      U     "IX_U_AXIS_ALM_CDE_BIT_3"; //E ;BOOL;U-Achse Alarm Bit 3
      =     "I_WK_ALARMCODE_BIT_3"; //M     374.3;BOOL;M-EINGANG: KometU-Achse:Alarmcode Bit 2e3

      U     "IX_U_AXIS_CONFIRM"; //E ;BOOL;U-Achse Quittierung
      =     "I_WK_QUIT_KOMMANDO"; //M     374.4;BOOL;M-EINGANG: KometU-Achse:Quit bei Pt

      U     "IX_U_AXIS_ALARM_N"; //E ;BOOL;U-Achse kein Alarm
      =     "I_WK_NEG_ALARM"; //M     374.5;BOOL;M-EINGANG: KometU-Achse:Alar

      U     "IX_U_AXIS_TOOL_ACTIVE_N"; //E ;BOOL;U-Achse keine Bearbeitung
      =     "I_WK_NEG_WZ_AKTIV"; //M     374.6;BOOL;M-EINGANG: KometU-Achse:Werkzeug beschäftig

      U     "IX_U_AXIS_TOOL_READY"; //E ;BOOL;U-Achse Werkzeug Betriebsbereit
      =     "I_WK_WZ_BTB"; //M     374.7;BOOL;M-EINGANG: KometU-Achse:System bereit

      U     "IX_U_AXIS_REF_SIGNAL"; //E ;BOOL;U-Achse Referenzimpuls
      =     "I_WK_REF"; //M     375.0;BOOL;M-EINGANG: KometU-Achse:RefNocken

      U     "IX_U_AXIS_READY"; //E ;BOOL;U-Achse Achse Betriebsbereit
      =     "I_WK_BTB"; //M     375.1;BOOL;M-EINGANG: KometU-Achse:Achse bereit

      U     "IX_U_AXIS_SWITCH_PLUS"; //E ;BOOL;U-Achse Endschalter positiv
      =     "I_WK_ENDSCHALTER_PLUS"; //M     375.2;BOOL;M-EINGANG: KometU-Achse:Vorendschalter positiv

      U     "IX_U_AXIS_SWITCH_MINUS"; //E ;BOOL;U-Achse Endschalter negativ
      =     "I_WK_ENDSCHALTER_MINUS"; //M     375.3;BOOL;M-EINGANG: KometU-Achse:Vorendschalter negativ
NETWORK
TITLE =Eingaenge Nicht verwendete Eingänge
//Eingänge, die in der HW konfiguriert werden müssen, aber noch nicht verwendet
//werden.
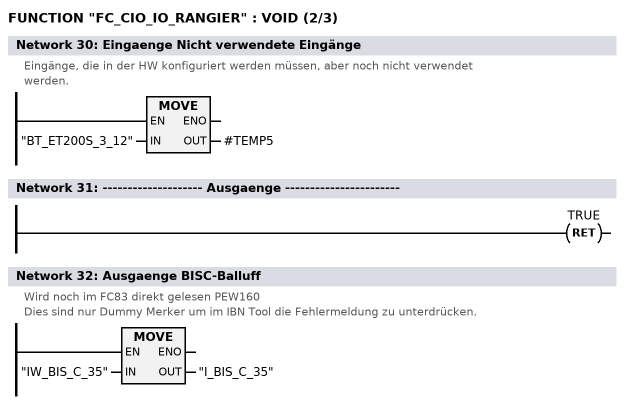
      L     "BT_ET200S_3_12"; //EW ;WORD;E5-03.5 Analogeingang Reserve
      T     #TEMP5;
NETWORK
TITLE =-------------------- Ausgaenge -----------------------

      BEA   ;

NETWORK
TITLE =Ausgaenge BISC-Balluff
//Wird noch im FC83 direkt gelesen PEW160
//Dies sind nur Dummy Merker um im IBN Tool die Fehlermeldung zu unterdrücken.
//
      L     "IW_BIS_C_35"; //PEW  1060;WORD;
      T     "I_BIS_C_35"; //MW    488;WORD;MW-EINGÄNGE:

NETWORK
TITLE =Ausgaenge allgemein
//Ausgänge
//
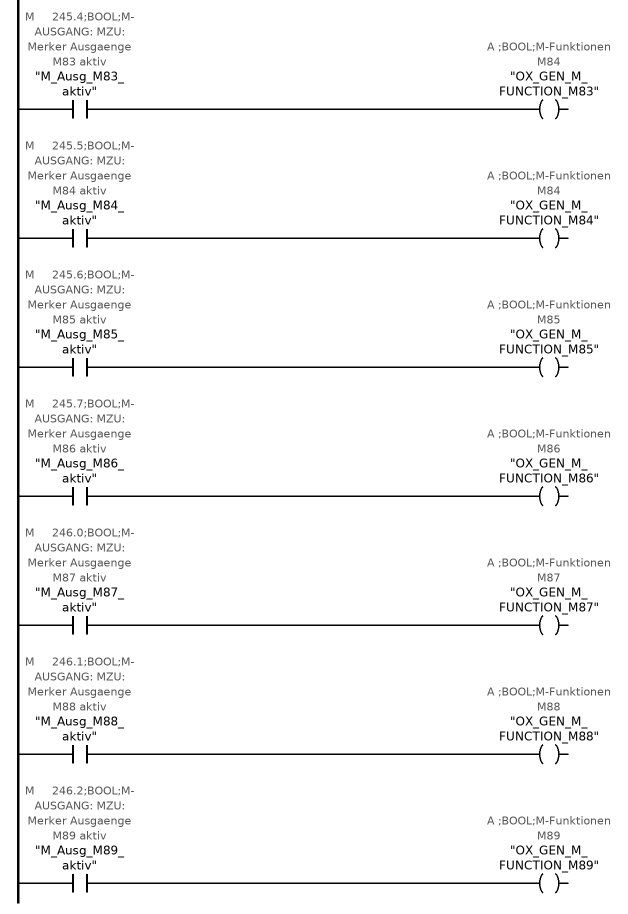
M003: NOP   0;

      U     "O_PW_FREIGABE"; //M     437.4;BOOL;M-AUSGANG: Anforderung Freigabe Palettenwechsel
      =     "OX_PC_ENABLE"; //A ;BOOL;Anforderung Freigabe Palettenwechsler   /G1-05.4

      U     "O_AL_PLC_BTB"; //M     432.1;BOOL;M-AUSGANG: Maschine 'Ein'  (CNC PLC Betriebsbereit)
      =     "OX_GEN_PLC_RDY"; //A ;BOOL;Maschine 'Ein'  (CNC PLC Betriebsbereit)

      U     "O_AL_Manual_Betrieb"; //M     432.2;BOOL;M-AUSGANG: Handbetrieb (Manual)
      =     "OX_AL_Manual_Betrieb"; //A ;BOOL;Handbetrieb (Manual)

      U     "O_GEN_CNC_PGM_ACTIVE"; //M     446.7;BOOL;M-AUSGANG: Betriebsstundenzaehler Programm laeuft
      =     "OX_GEN_CNC_PGM_ACTIVE"; //A ;BOOL;Betriebsstundenzaehler Programm laeuft

      U     "O_AL_XACHS_Bremse_auf"; //M     140.1;BOOL;M-AUSGANG: Ansteuerung Motorbremse X-Achse
      =     "OX_AL_XACHS_Bremse_auf"; //A ;BOOL;Ansteuerung Motorbremse X-Achse

      U     "O_AL_YACHS_Bremse_auf"; //M     140.3;BOOL;M-AUSGANG: Ansteuerung Motorbremse Y-Achse
      =     "OX_AL_YACHS_Bremse_auf"; //A ;BOOL;Ansteuerung Motorbremse Y-Achse

      U     "O_AL_ZACHS_Bremse_auf"; //M     140.5;BOOL;M-AUSGANG: Ansteuerung Motorbremse Z-Achse
      =     "OX_AL_ZACHS_Bremse_auf"; //A ;BOOL;Ansteuerung Motorbremse Z-Achse

      U     "O_AL_4ACHS_Bremse_auf"; //M     140.7;BOOL;M-AUSGANG: Ansteuerung Motorbremse 4-Achse
      =     "OX_AL_4ACHS_Bremse_auf"; //A ;BOOL;Ansteuerung Motorbremse 4-Achse

      U     "O_AL_5ACHS_Bremse_auf"; //M     141.1;BOOL;M-AUSGANG: Ansteuerung Motorbremse 5-Achse
      =     "OX_AL_5ACHS_Bremse_auf"; //A ;BOOL;Ansteuerung Motorbremse 5-Achse

      UN    "O_4_Klem_Bremse_Auf"; //M     433.5;BOOL;M-AUSGANG: 4.Achse Klemmung lösen
      =     "OX_AL_4ACHS_Klemmen"; //A ;BOOL;4.Achse klemmen

      UN    "O_5_Klem_Bremse_Auf"; //M     433.6;BOOL;M-AUSGANG: 5.Achse Klemmung lösen
      =     "OX_GEN_AXIS5_CLAMP"; //A ;BOOL;5.Achse klemmen

      UN    "O_5_Klem_Bremse_Auf"; //M     433.6;BOOL;M-AUSGANG: 5.Achse Klemmung lösen
      =     "OX_DH_CLAMP_RELEASE"; //A ;BOOL;Klemmung loesen NC-Teilapparat

      U     "M_SBH_AKTIV_ARBEITSRAUM"; //M     539.0;BOOL;SAFETY: SBH aktiv -> Freigabe Arbeitsraumtüre entriegeln
      =     "OX_GEN_CABIN_UNLOCK"; //A ;BOOL;Magnetverriegelung Kabinentüre entriegeln

      U     "O_AL_Hydraulik_Ein"; //M     433.3;BOOL;M-AUSGANG: Hydraulik 'Ein'
      =     "OX_GEN_HYD_ON"; //A ;BOOL;Hydraulik 'Ein'

      U     "O_AL_Druckluft_ein"; //M     433.2;BOOL;M-AUSGANG: Pneumatik 'Ein'
      =     "OX_GEN_CAIR_ON"; //A ;BOOL;Pneumatik 'Ein'

      U     "O_AL_Blasluft_M25"; //M     439.4;BOOL;M-AUSGANG: Blasluft Kuehlung Werkzeug 'Ein'
      =     "OX_SPI_CAIR_JETS_EXT"; //A ;BOOL;Blasluft Kuehlung Werkzeug 'Ein'

      U     "O_AL_4_BA_Selbsthaltung"; //M     437.7;BOOL;M-AUSGANG: Energiefreigabe 4.Betriebsart
      =     "OX_GEN_OM_4_ENABLE"; //A ;BOOL;Energiefreigabe 4.Betriebsart

      U     "O_AL_SCH_Pumpe_ein"; //M     432.4;BOOL;M-AUSGANG: Schmierung Maschine 'Ein'
      =     "OX_GEN_LUB_ON"; //A ;BOOL;Schmierung Maschine 'Ein'

      U     "O_AL_SCH_M26_Pumpe_ein"; //M     451.1;BOOL;M-AUSGANG: Dreh-Duchführung Ansteuerung Schmierpumpe 'Ein'
      =     "OX_SPI_ROTRA_LUB_ON"; //A ;BOOL;Dreh-Duchführung Ansteuerung Schmierpumpe 'Ein'

      U     "O_WZ_MIN_SCH_Ums_M7"; //M     104.7;BOOL;M-AUSGANG: Umschaltung Ventil Schmiersystem innere Kuehlmittelzufuhr
      =     "OX_TOOL_MQL_M7"; //A ;BOOL;Umschaltung Ventil Schmiersystem innere Kuehlmittelzufuhr

      U     "O_WZ_MIN_SCH_MV2"; //M      83.3;BOOL;M-AUSGANG: Minimalmengen Schmierung Ventil 2 Ein
      =     "OX_TOOL_MQL_VAL_2"; //A ;BOOL;Minimalmengen Schmierung Ventil 2 Ein

      U     "O_WZ_MIN_SCH_MV1"; //M     450.7;BOOL;M-AUSGANG: Minimalmengen Schmierung Ventil 1 Ein
      =     "OX_TOOL_MQL_VAL_1"; //A ;BOOL;Minimalmengen Schmierung Ventil 1 Ein

      U     "O_WZ_MIN_SCH_Ums_M8"; //M     104.2;BOOL;M-AUSGANG: Umschaltung Ventil Schmiersystem Kuehlmittel 1
      =     "OX_TOOL_MQL_M8"; //A ;BOOL;Umschaltung Ventil Schmiersystem Kuehlmittel 1

      U     "O_AL_Tempkomp_DSR"; //M     432.5;BOOL;M-AUSGANG: Temperaturkompensation rücksetzen Synchronisation Temperaturdaten
      =     "OX_AL_Tempkomp_DSR"; //A ;BOOL;TEMPERATURKOMPENSATION: rücksetzen Synchronisation Temperaturdaten

      U     "O_AL_Tempkomp_CTS"; //M     432.6;BOOL;M-AUSGANG: Temperaturkompensation   Temperaturdaten auslesen
      =     "OX_AL_Tempkomp_CTS"; //A ;BOOL;TEMPERATURKOMPENSATION: Temperaturdaten auslesen

      U     "O_AL_LM_RD"; //M     327.0;BOOL;M-AUSGANG: Signalleuchte Farbe RD
      =     "OX_GEN_SIGNALLAMP_RD"; //A ;BOOL;Signalleuchte Farbe RD

      U     "O_AL_LM_GN"; //M     327.2;BOOL;M-AUSGANG: Signalleuchte Farbe GN
      =     "OX_GEN_SIGNALLAMP_GN"; //A ;BOOL;Signalleuchte Farbe GN

      U     "O_AL_LM_YE"; //M     327.1;BOOL;M-AUSGANG: Signalleuchte Farbe YE
      =     "OX_GEN_SIGNALLAMP_YE"; //A ;BOOL;Signalleuchte Farbe YE

      U     "O_AL_LM_BU"; //M     327.3;BOOL;M-AUSGANG: Signalleuchte Farbe BU
      =     "OX_GEN_SIGNALLAMP_BU"; //A ;BOOL;Signalleuchte Farbe BU

      U     "O_GEN_OM_ID_DATA_0"; //M     446.5;BOOL;M-AUSGANG: Smartkey -  Rückmeldung Daten-Spur 1
      =     "OX_GEN_OM_ID_DATA_0"; //A ;BOOL;Smartkey: Rückmeldung Daten – Spur 1

      U     "O_GEN_OM_ID_DATA_1"; //M     446.6;BOOL;M-AUSGANG: Smartkey -  Rückmeldung Daten-Spur 2
      =     "OX_GEN_OM_ID_DATA_1"; //A ;BOOL;Smartkey: Rückmeldung Daten – Spur 2

      U     "O_GEN_OPTWAVE_GN"; //M    2061.2;BOOL;M-AUSGANG: Signalband Farbe Grün
      =     "OX_GEN_OPTWAVE_GN"; //A ;BOOL;Signalband neues Design Farbe GN

      U     "O_GEN_OPTWAVE_RD"; //M    2061.0;BOOL;M-AUSGANG: Signalband Farbe Rot
      =     "OX_GEN_OPTWAVE_RD"; //A ;BOOL;Signalband neues Design Farbe RD

      U     "O_GEN_OPTWAVE_BU"; //M    2061.3;BOOL;M-AUSGANG: Signalband Farbe Blau
      =     "OX_GEN_OPTWAVE_BU"; //A ;BOOL;Signalband neues Design Farbe  BU

      U     "O_AL_Start_Sig_Renishaw"; //M     433.7;BOOL;M-AUSGANG: Messtasterfreigabe
      =     "OX_AL_Start_Sig_Renishaw"; //A ;BOOL;Messtasterfreigabe

      U     "O_AL_Start_Sig_Renishaw"; //M     433.7;BOOL;M-AUSGANG: Messtasterfreigabe
      =     "OX_TP_ENABLE"; //A ;BOOL;Startsignal Messtaster

      U     "O_AL_NEBELABSCH_EIN"; //M     113.6;BOOL;M-AUSGANG: Nebel- u.Rauchabscheider 'Ein'
      =     "OX_OMS_ON"; //A ;BOOL;Nebel- u.Rauchabscheider 'Ein'

      U     "O_AL_NEG_POWERSAVE_STBY"; //M     344.7;BOOL;M-AUSGANG: Maschinenabschaltung
      =     "OX_GEN_POWERSAVE_N"; //A ;BOOL;Maschinenabschaltung

      U     "O_PW_SPANNDRUCK_HYD_AUS"; //M     436.3;BOOL;M-AUSGANG: MA H4-03.7 Spannvorrichtung Verriegelung Palettenwechsler
      =     "OX_PC_CL_PRESS_HYD_OFF"; //A ;BOOL;MA H4-03.7 Spannvorrichtung Verriegelung Palettenwechs

      U     "O_Funktion_M20"; //M     435.6;BOOL;M-AUSGANG: Zusatzfunktion M190
      =     "OX_AL_Funktion_M20"; //A ;BOOL;M-Funktionen M190

      U     "M_Ausg_M80_aktiv"; //M     245.1;BOOL;M-AUSGANG: MZU: Merker Ausgaenge M80 aktiv
      =     "OX_GEN_M_FUNCTION_M80"; //A ;BOOL;M-Funktionen M80

      U     "M_Ausg_M81_aktiv"; //M     245.2;BOOL;M-AUSGANG: MZU: Merker Ausgaenge M81 aktiv
      =     "OX_GEN_M_FUNCTION_M81"; //A ;BOOL;M-Funktionen M81

      U     "M_Ausg_M82_aktiv"; //M     245.3;BOOL;M-AUSGANG: MZU: Merker Ausgaenge M82 aktiv
      =     "OX_GEN_M_FUNCTION_M82"; //A ;BOOL;M-Funktionen M82

      U     "M_Ausg_M83_aktiv"; //M     245.4;BOOL;M-AUSGANG: MZU: Merker Ausgaenge M83 aktiv
      =     "OX_GEN_M_FUNCTION_M83"; //A ;BOOL;M-Funktionen M84

      U     "M_Ausg_M84_aktiv"; //M     245.5;BOOL;M-AUSGANG: MZU: Merker Ausgaenge M84 aktiv
      =     "OX_GEN_M_FUNCTION_M84"; //A ;BOOL;M-Funktionen M84

      U     "M_Ausg_M85_aktiv"; //M     245.6;BOOL;M-AUSGANG: MZU: Merker Ausgaenge M85 aktiv
      =     "OX_GEN_M_FUNCTION_M85"; //A ;BOOL;M-Funktionen M85

      U     "M_Ausg_M86_aktiv"; //M     245.7;BOOL;M-AUSGANG: MZU: Merker Ausgaenge M86 aktiv
      =     "OX_GEN_M_FUNCTION_M86"; //A ;BOOL;M-Funktionen M86

      U     "M_Ausg_M87_aktiv"; //M     246.0;BOOL;M-AUSGANG: MZU: Merker Ausgaenge M87 aktiv
      =     "OX_GEN_M_FUNCTION_M87"; //A ;BOOL;M-Funktionen M87

      U     "M_Ausg_M88_aktiv"; //M     246.1;BOOL;M-AUSGANG: MZU: Merker Ausgaenge M88 aktiv
      =     "OX_GEN_M_FUNCTION_M88"; //A ;BOOL;M-Funktionen M88

      U     "M_Ausg_M89_aktiv"; //M     246.2;BOOL;M-AUSGANG: MZU: Merker Ausgaenge M89 aktiv
      =     "OX_GEN_M_FUNCTION_M89"; //A ;BOOL;M-Funktionen M89
NETWORK
TITLE =Ausgänge für Vibrationssensor

      L     "DB_PLC_MD_DB20".UDInt._044_ANWAHL_VIBRATIONSEN;
      L     1;
      >=I   ;
      SPBN  kVMS;

      L     "MW_VMS_SPI_SPEED_RPM"; //MW    612;INT;Analogausgang Vibrationssensor Spindeldrehzahl
      T     "OW_VMS_SPI_SPEED_RPM"; //AW ;WORD;

      U     "O_VMS_MSG_BEA_START"; //M     671.2;BOOL;
      =     "OX_VMS_MSG_BEA_START"; //A ;BOOL;

kVMS: NOP   0;
NETWORK
TITLE =Ausgaenge an NCU und NC Baugruppe SOLUTIONLINE
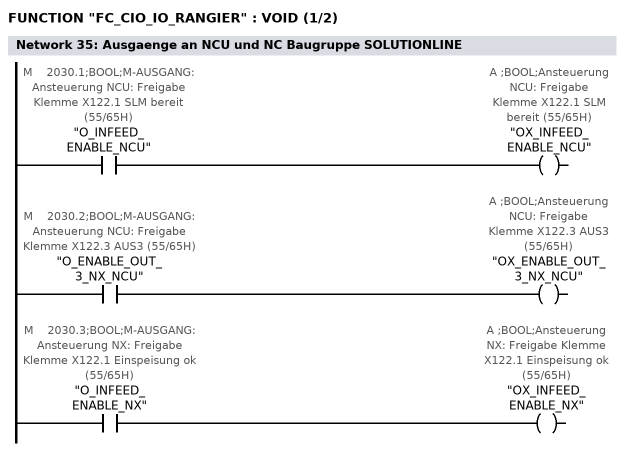

      NOP   0;

      U     "O_INFEED_ENABLE_NCU"; //M    2030.1;BOOL;M-AUSGANG: Ansteuerung NCU: Freigabe Klemme X122.1 SLM bereit (55/65H)
      =     "OX_INFEED_ENABLE_NCU"; //A ;BOOL;Ansteuerung NCU: Freigabe Klemme X122.1 SLM bereit (55/65H)

      U     "O_ENABLE_OUT_3_NX_NCU"; //M    2030.2;BOOL;M-AUSGANG: Ansteuerung NCU: Freigabe Klemme X122.3 AUS3 (55/65H)
      =     "OX_ENABLE_OUT_3_NX_NCU"; //A ;BOOL;Ansteuerung NCU: Freigabe Klemme X122.3 AUS3 (55/65H)

      U     "O_INFEED_ENABLE_NX"; //M    2030.3;BOOL;M-AUSGANG: Ansteuerung NX: Freigabe Klemme X122.1 Einspeisung ok (55/65H)
      =     "OX_INFEED_ENABLE_NX"; //A ;BOOL;Ansteuerung NX: Freigabe Klemme X122.1 Einspeisung ok (55/65H)
NETWORK
TITLE =Ausgaenge Schwenkkopf und Spindel
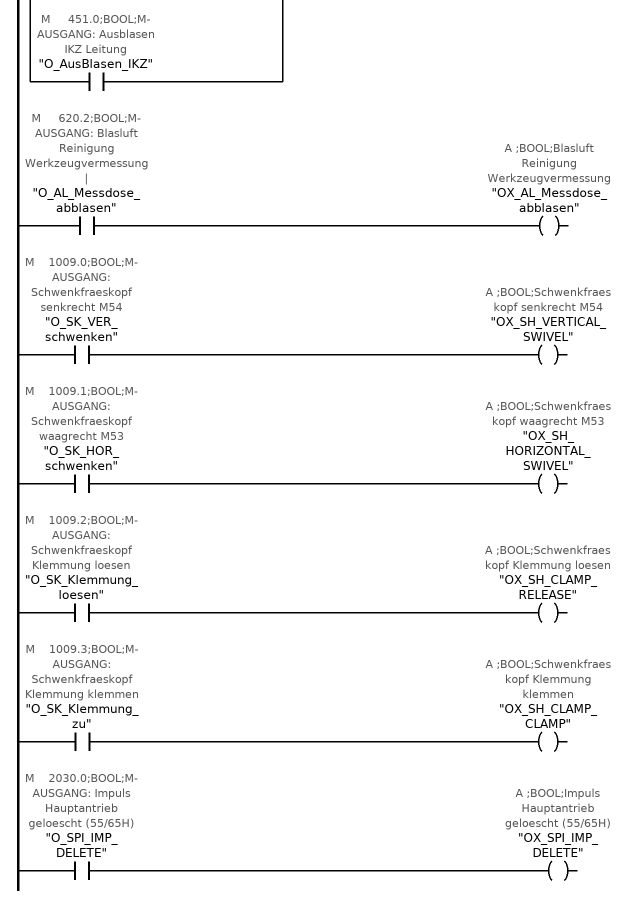

      U     "O_SPI_klemmen"; //M     283.1;BOOL;M-AUSGANG: Fraesspindel klemmen
      =     "OX_SPI_CLAMP"; //A ;BOOL;Fraesspindel klemmen

      U     "O_SPI_loesen"; //M     283.2;BOOL;M-AUSGANG: Fraesspindel loesen
      =     "OX_SPI_RELEASE"; //A ;BOOL;Fraesspindel loesen

      U     "O_Y_Umschaltung_SPI"; //M     447.1;BOOL;M-AUSGANG: Stern Dreieck: Ausgang Stern
      =     "OX_SPI_WYE"; //A ;BOOL;Stern Dreieck: Ausgang Stern

      U     "O_D_Umschaltung_SPI"; //M     447.2;BOOL;M-AUSGANG: Stern Dreieck: Ausgang Dreieck
      =     "OX_SPI_DELTA"; //A ;BOOL;Stern Dreieck: Ausgang Dreieck

      U     "O_SK_1_Stufe_Getriebe"; //M     433.0;BOOL;M-AUSGANG: Drehzahlschaltung Hauptantrieb mit Getriebe    Drehzahl kleiner
      =     "OX_SH_GEAR_STAGE1"; //A ;BOOL;Drehzahlschaltung Hauptantrieb mit Getriebe    Drehzahl kle

      U     "O_SK_2_Stufe_Getriebe"; //M     433.1;BOOL;M-AUSGANG: Drehzahlschaltung Hauptantrieb mit Getriebe    Drehzahl größer
      =     "OX_SH_GEAR_STAGE2"; //A ;BOOL;Drehzahlschaltung Hauptantrieb mit Getriebe    Drehzahl gr

      U     "O_SPI_SCH_LUFT"; //M     435.1;BOOL;M-AUSGANG: Schwenkfräskopf Druckluft Schmierung 'Ein'
      =     "OX_SPI_LUB_CAIR_ON"; //A ;BOOL;Schwenkfräskopf Druckluft Schmierung 'Ein'

      U     "O_SPI_SCH_OEL"; //M     435.0;BOOL;M-AUSGANG: Schmierung Hauptantrieb 24.000 U/min
      =     "OX_SPI_LUB_OIL_PUMP_ON"; //A ;BOOL;Schmierung Hauptantrieb 24.000 U/min

      U     "O_WZKegel_Blasluft"; //M     434.0;BOOL;M-AUSGANG: Messtaster Messstelle reinigen (M29) und  Werkzeugkegel ausblasen
      O(    ;
      U     "O_Blasluft_Messtaster"; //M     440.3;BOOL;M-AUSGANG: Blasluft Messtaster
      UN    "M_24aktiv"; //M     214.3;BOOL;LA: Laser ausfahren M24 aktiv
      )     ;
      O     "O_M7_Luftkuehlung"; //M     443.4;BOOL;M-AUSGANG: M7 Luftkuehlung
      O     "O_AusBlasen_IKZ"; //M     451.0;BOOL;M-AUSGANG: Ausblasen IKZ Leitung
      =     "OX_SPI_CAIR_TOOL"; //A ;BOOL;Druckluft Werkzeugkegel ausblasen

      U     "O_AL_Messdose_abblasen"; //M     620.2;BOOL;M-AUSGANG: Blasluft Reinigung Werkzeugvermessung |
      =     "OX_AL_Messdose_abblasen"; //A ;BOOL;Blasluft Reinigung Werkzeugvermessung

      U     "O_SK_VER_schwenken"; //M    1009.0;BOOL;M-AUSGANG: Schwenkfraeskopf senkrecht M54
      =     "OX_SH_VERTICAL_SWIVEL"; //A ;BOOL;Schwenkfraeskopf senkrecht M54

      U     "O_SK_HOR_schwenken"; //M    1009.1;BOOL;M-AUSGANG: Schwenkfraeskopf waagrecht M53
      =     "OX_SH_HORIZONTAL_SWIVEL"; //A ;BOOL;Schwenkfraeskopf waagrecht M53

      U     "O_SK_Klemmung_loesen"; //M    1009.2;BOOL;M-AUSGANG: Schwenkfraeskopf Klemmung loesen
      =     "OX_SH_CLAMP_RELEASE"; //A ;BOOL;Schwenkfraeskopf Klemmung loesen

      U     "O_SK_Klemmung_zu"; //M    1009.3;BOOL;M-AUSGANG: Schwenkfraeskopf Klemmung klemmen
      =     "OX_SH_CLAMP_CLAMP"; //A ;BOOL;Schwenkfraeskopf Klemmung klemmen

      U     "O_SPI_IMP_DELETE"; //M    2030.0;BOOL;M-AUSGANG: Impuls Hauptantrieb geloescht (55/65H)
      =     "OX_SPI_IMP_DELETE"; //A ;BOOL;Impuls Hauptantrieb geloescht (55/65H)

NETWORK
TITLE =Ausgänge WZ-Spanner

//Bei H-Maschinen werdem die Ausgänge durch den OB35 Aufruf geschrieben (Span_zu_Span_Zeit Optimierung)
      U     "DB_CONFIG".ANWAHL_DURCH_USER_DATA.MASCHTYP_3071_AKTIV;
      SPB   Hma2;

      U     "O_AL_WZ_Spanner_Loesen"; //M     433.4;BOOL;M-AUSGANG: Werkzeugspanner lösen (Autobetr)/Anwahl lösen (Handbetr)
      O     "M_O_Anwahl_WZS_Man"; //M     195.5;BOOL;WSP: Ausgang Manuelles loesen Spanner
      =     "OX_SPI_TL_CLAMP_RELEASE"; //A ;BOOL;Werkzeugspanner loesen

      UN    "O_AL_WZ_Spanner_Loesen"; //M     433.4;BOOL;M-AUSGANG: Werkzeugspanner lösen (Autobetr)/Anwahl lösen (Handbetr)
      UN    "M_Tast_Man_WZSp"; //M     386.0;BOOL;WZ-SPANNER:Werkzeugspanner manuell lösen
      =     "OX_SPI_TL_CLP_CLAMP"; //A ;BOOL;Werkzeugspanner spannen

Hma2: NOP   0;
NETWORK
TITLE =Ausgaenge Handrad
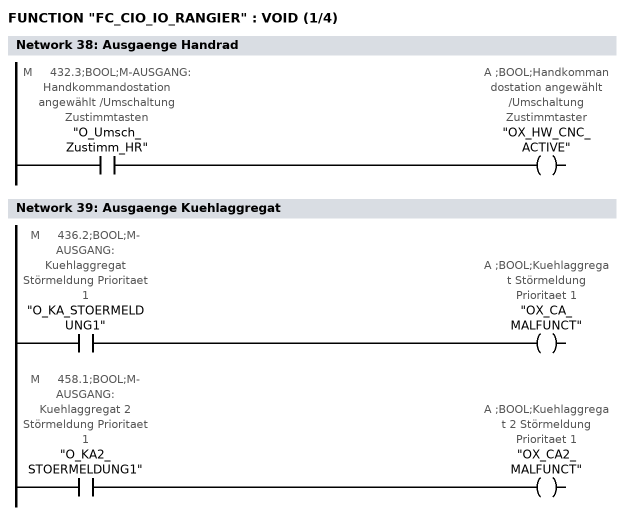

      NOP   0;

      U     "O_Umsch_Zustimm_HR"; //M     432.3;BOOL;M-AUSGANG: Handkommandostation angewählt /Umschaltung Zustimmtasten
      =     "OX_HW_CNC_ACTIVE"; //A ;BOOL;Handkommandostation angewählt /Umschaltung Zustimmtaster

NETWORK
TITLE =Ausgaenge Kuehlaggregat

      NOP   0;

      U     "O_KA_STOERMELDUNG1"; //M     436.2;BOOL;M-AUSGANG: Kuehlaggregat Störmeldung Prioritaet 1
      =     "OX_CA_MALFUNCT"; //A ;BOOL;Kuehlaggregat Störmeldung Prioritaet 1

      U     "O_KA2_STOERMELDUNG1"; //M     458.1;BOOL;M-AUSGANG: Kuehlaggregat 2 Störmeldung Prioritaet 1
      =     "OX_CA2_MALFUNCT"; //A ;BOOL;Kuehlaggregat 2 Störmeldung Prioritaet 1
NETWORK
TITLE =Ausgaenge Spannhydraulik
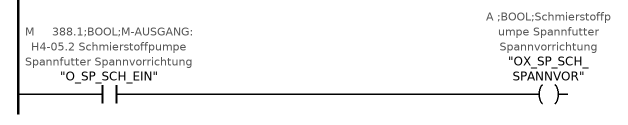

      NOP   0;

      U     "O_SP_HYD_EIN"; //M     458.3;BOOL;M-AUSGANG: Spannhydraulik Pumpe ein
      =     "OX_HCD_ON"; //A ;BOOL;Spannhydraulik ein   /H4-01.6

      U     "O_SP_HYD_RPL_LOESEDR_OK"; //M     382.0;BOOL;M-AUSGANG: Spannvorrichtung Loesedruck vorhanden
      =     "OX_HCD_CL_PR_SST_RELD_H"; //A ;BOOL;Spannhydraulik Leuchtmelder Vorrichtung entspannen   /H4-10.6

      U     "O_SP_HYD_RPL_SPANNDR_OK"; //M     382.1;BOOL;M-AUSGANG: Spannvorrichtung Spanndruck vorhanden
      =     "OX_HCD_CL_PR_SST_CLPED_H"; //A ;BOOL;Spannhydraulik Leuchtmelder Vorrichtung spannen   /H4-10.3

      U     "O_SP_H_SPANNSTELLE_1"; //M     356.0;BOOL;M-AUSGANG: Spannhydraulik Lampe Spannstelle 1
      =     "OX_HCD_SST_CL_PO_1_SEL_H"; //A ;BOOL;Spannhydraulik Rüstplatz Leuchtmelder Spannstelle 1 aktiv   /H4-50.3

      U     "O_SP_H_SPANNSTELLE_2"; //M     356.1;BOOL;M-AUSGANG: Spannhydraulik Lampe Spannstelle 2
      =     "OX_HCD_SST_CL_PO_2_SEL_H"; //A ;BOOL;Spannhydraulik Rüstplatz Leuchtmelder Spannstelle 2 aktiv   /H4-50.6

      U     "O_SP_H_SPANNSTELLE_3"; //M     356.2;BOOL;M-AUSGANG: Spannhydraulik Lampe Spannstelle 3
      =     "OX_SP_H_SPANNSTELLE_3"; //A ;BOOL;Spannhydraulik Lampe Spannstelle 3

      U     "O_SP_H_SPANNSTELLE_4"; //M     356.3;BOOL;M-AUSGANG: Spannhydraulik Lampe Spannstelle 4
      =     "OX_SP_H_SPANNSTELLE_4"; //A ;BOOL;Spannhydraulik Lampe Spannstelle 4

      U     "O_SST_FIXT_CL_PO_1_CLE"; //M     384.6;BOOL;MA H4-94.2 Auflagenkontrolle Luft für Reinigung (hoher ALK-Druck)
      =     "OX_SST_FIXT_CL_PO_1_CLE"; //A ;BOOL;H4-94.2 Auflagenkontrolle Luft für Reinigung (hoher ALK-Druck)

      U     "O_SST_SC_SENS_ACT"; //M     384.7;BOOL;MA H4-94.4 Auflagenkontrolle Luft für Messung (niedriger ALK-Druck)
      =     "OX_SST_SC_SENS_ACT"; //A ;BOOL;H4-94.4 Auflagenkontrolle Luft für Messung (niedriger ALK-Druck)

      U     "O_SST_SC_CL_PO_1_STATE"; //M     379.4;BOOL;MA H4-93.2 Status Auflagenkontrolle Spannstelle 1 (Meldeleuchte)
      =     "OX_SST_SC_CL_PO_1_STATE"; //A ;BOOL;H4-93.2 Status Auflagenkontrolle Spannstelle 1 (Meldeleuchte)

      U     "O_SST_SC_CL_PO_2_STATE"; //M     379.5;BOOL;MA H4-93.4 Status Auflagenkontrolle Spannstelle 2 (Meldeleuchte)
      =     "OX_SST_SC_CL_PO_2_STATE"; //A ;BOOL;H4-93.4 Status Auflagenkontrolle Spannstelle 2 (Meldeleuchte)

      U     "O_SP_RPL_BLASLUFT"; //M     357.7;BOOL;M-AUSGANG: Ventil Luft für Vorrichtung Abblasen
      =     "OX_HCD_SST_BLOW_AIR"; //A ;BOOL;Medienkupplung Ruestplatz abblasen

      U     "O_SP_MPL_BLASLUFT"; //M     205.7;BOOL;M-AUSGANG: Blasluft Medienkupplung Spannhydraulik 'Ein'
      =     "OX_HCD_TST_MCON_CLEAN"; //A ;BOOL;Hydraulik Maschinenplatz Kupplung abblasen   /H4-08.2

      U     "O_SP_RPL_MPL_BLASLUFT"; //M      24.6;BOOL;M-AUSGANG: Ventil Blasluft Medienkupplung
      =     "OX_SP_RPL_MPL_BLASLUFT"; //A ;BOOL;Ventil Blasluft Medienkupplung

      U     "O_SP_SCH_EIN"; //M     388.1;BOOL;M-AUSGANG: H4-05.2 Schmierstoffpumpe Spannfutter Spannvorrichtung
      =     "OX_HCD_LUB_ON"; //A ;BOOL;

      U     "O_SP_RPL_DRUCKLOS"; //M     387.5;BOOL;M-AUSGANG: Ruestplatz Ventil Drucklos
      =     "OX_HCD_SST_UNPRESS"; //A ;BOOL;Ruestplatz Ventil Drucklos

      U     "O_SP_RPL_DRUCK_AUS"; //M     357.4;BOOL;M-AUSGANG: H4-29.1 Spanndruck Rüstplatz Aus
      =     "OX_HCD_SST_PRESSURE_OFF"; //A ;BOOL;

      U     "O_SP_RPL_GESPANNT"; //M     387.4;BOOL;M-AUSGANG: Spannhydraulik Ruestplatz gespannt
      =     "OX_HCD_SST_LOCK"; //A ;BOOL;Spannhydraulik Ruestplatz gespannt

      U     "O_SP_RPL_SPANNEN"; //M     387.7;BOOL;Spannhydraulik Ruestplatz spannen
      =     "OX_HCD_SST_CLAMP"; //A ;BOOL;Spannhydraulik Ruestplatz spannen

      U     "O_SP_MPL_DRU_OK"; //M     387.6;BOOL;M-AUSGANG: Spannvorrichtung Maschine gespannt
      =     "OX_HCD_MPL_PRESSURE_OK"; //A ;BOOL;Spannvorrichtung Maschine gespannt

      U     "O_SP_MASCHINE_ENTLADEN"; //M     388.0;BOOL;M-AUSGANG: H4-07.6 Rueckmeldung Maschine Entladen
      =     "OX_HCD_MACHINE_UNLOAD"; //A ;BOOL;Rueckmeldung Maschine Entladen

      U     "O_SP_SCH_EIN"; //M     388.1;BOOL;M-AUSGANG: H4-05.2 Schmierstoffpumpe Spannfutter Spannvorrichtung
      =     "OX_SP_SCH_SPANNVOR"; //A ;BOOL;Schmierstoffpumpe Spannfutter Spannvorrichtung

NETWORK
TITLE =Ausgaenge ProfiBus: HAWE-Box
//PABs müssen ABSOLUT sein, da IBN-Tool PAB-Symbole nicht verarbeitet
//-----------------------------------------------------------------------------
//
//      U     "m_null"
//      =     L     16.0
//      BLD   103
//      U     "m_eins"
//      =     L     16.1
//      BLD   103
//      U     "DB_HR".ABST.SpannHydraulik
//      UN    "DB_HR".ABST.SP_vorbereitet
//      SPBNB _003
//      CALL  "FC_UT_IO_PROFIBUS"
//       read        :=L16.0
//       write       :=L16.1
//       Datenbereich:="DB_HR".HAWE.an
//       Profibus_ADR:=430
//_003: NOP   0
//
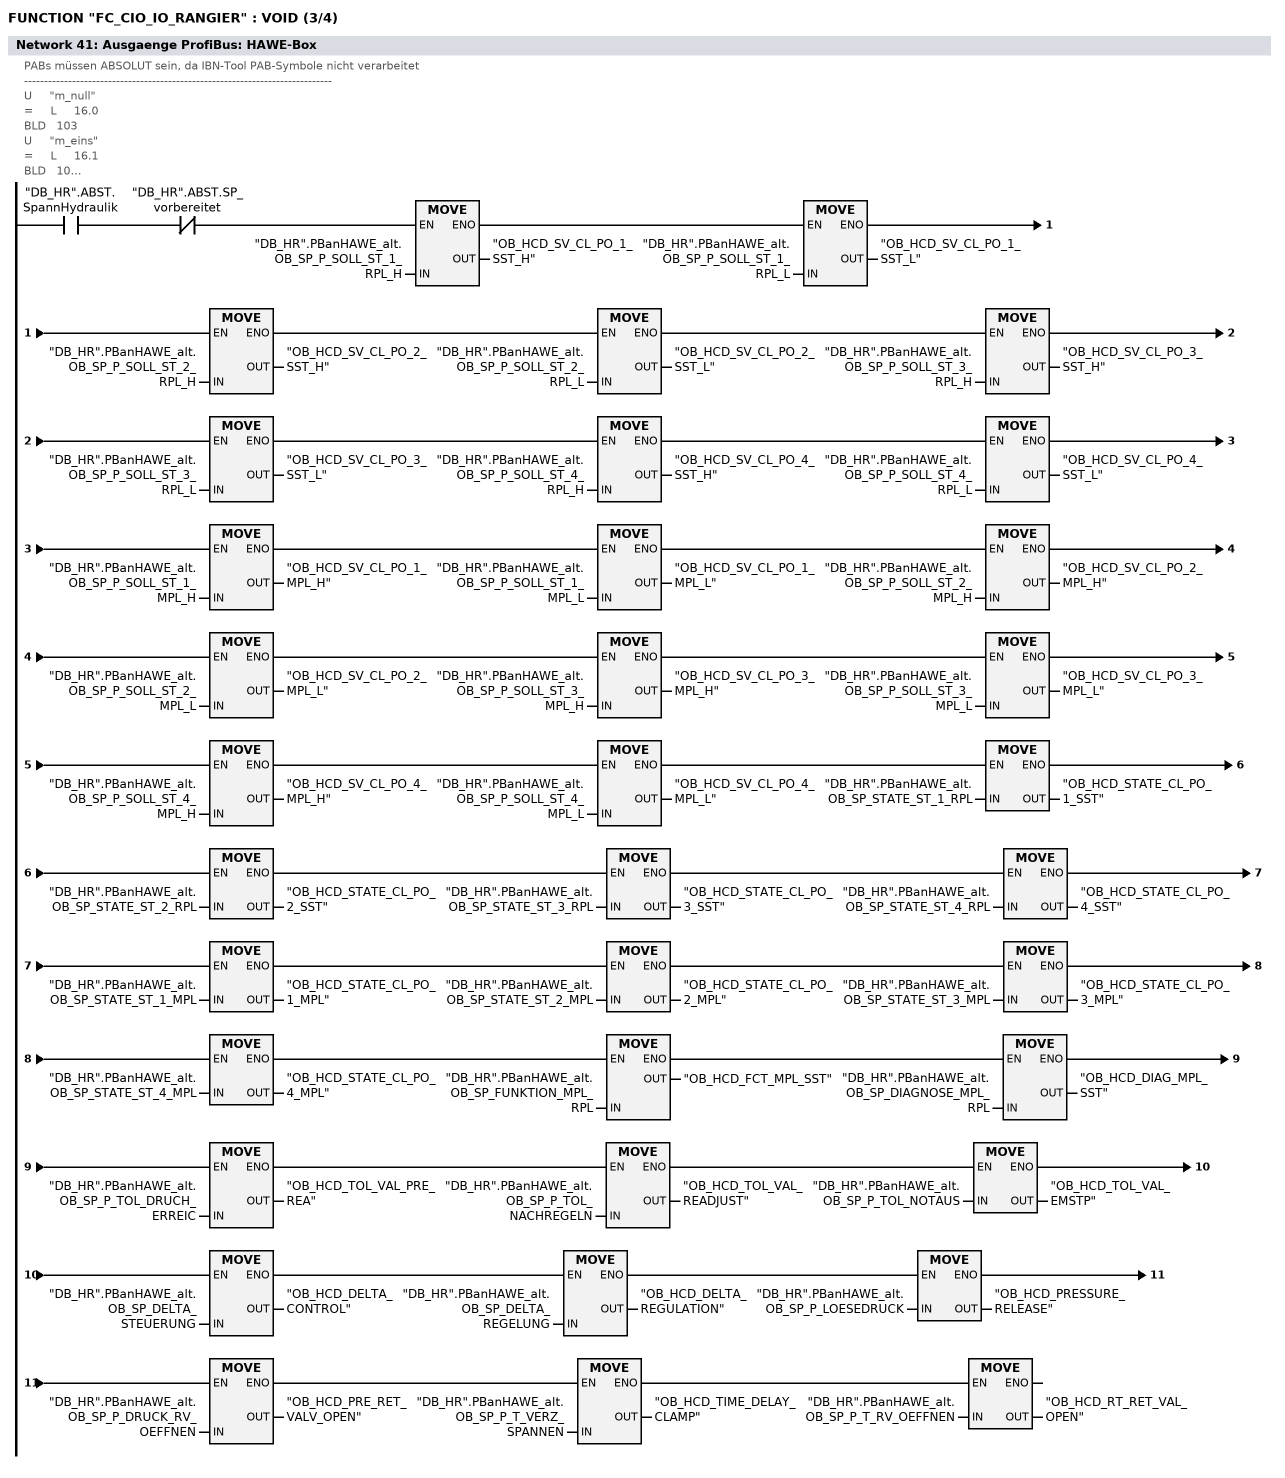
      U     "DB_HR".ABST.SpannHydraulik;
      UN    "DB_HR".ABST.SP_vorbereitet;
      SPBN  khw;

      L     "DB_HR".PBanHAWE_alt.OB_SP_P_SOLL_ST_1_RPL_H;
      T     "OB_HCD_SV_CL_PO_1_SST_H"; //PAB   430;BYTE;

      L     "DB_HR".PBanHAWE_alt.OB_SP_P_SOLL_ST_1_RPL_L;
      T     "OB_HCD_SV_CL_PO_1_SST_L"; //PAB   431;BYTE;

      L     "DB_HR".PBanHAWE_alt.OB_SP_P_SOLL_ST_2_RPL_H;
      T     "OB_HCD_SV_CL_PO_2_SST_H"; //PAB   432;BYTE;

      L     "DB_HR".PBanHAWE_alt.OB_SP_P_SOLL_ST_2_RPL_L;
      T     "OB_HCD_SV_CL_PO_2_SST_L"; //PAB   433;BYTE;

      L     "DB_HR".PBanHAWE_alt.OB_SP_P_SOLL_ST_3_RPL_H;
      T     "OB_HCD_SV_CL_PO_3_SST_H"; //PAB   434;BYTE;

      L     "DB_HR".PBanHAWE_alt.OB_SP_P_SOLL_ST_3_RPL_L;
      T     "OB_HCD_SV_CL_PO_3_SST_L"; //PAB   435;BYTE;

      L     "DB_HR".PBanHAWE_alt.OB_SP_P_SOLL_ST_4_RPL_H;
      T     "OB_HCD_SV_CL_PO_4_SST_H"; //PAB   436;BYTE;

      L     "DB_HR".PBanHAWE_alt.OB_SP_P_SOLL_ST_4_RPL_L;
      T     "OB_HCD_SV_CL_PO_4_SST_L"; //PAB   437;BYTE;

      L     "DB_HR".PBanHAWE_alt.OB_SP_P_SOLL_ST_1_MPL_H;
      T     "OB_HCD_SV_CL_PO_1_MPL_H"; //PAB   438;BYTE;

      L     "DB_HR".PBanHAWE_alt.OB_SP_P_SOLL_ST_1_MPL_L;
      T     "OB_HCD_SV_CL_PO_1_MPL_L"; //PAB   439;BYTE;

      L     "DB_HR".PBanHAWE_alt.OB_SP_P_SOLL_ST_2_MPL_H;
      T     "OB_HCD_SV_CL_PO_2_MPL_H"; //PAB   440;BYTE;

      L     "DB_HR".PBanHAWE_alt.OB_SP_P_SOLL_ST_2_MPL_L;
      T     "OB_HCD_SV_CL_PO_2_MPL_L"; //PAB   441;BYTE;

      L     "DB_HR".PBanHAWE_alt.OB_SP_P_SOLL_ST_3_MPL_H;
      T     "OB_HCD_SV_CL_PO_3_MPL_H"; //PAB   442;BYTE;

      L     "DB_HR".PBanHAWE_alt.OB_SP_P_SOLL_ST_3_MPL_L;
      T     "OB_HCD_SV_CL_PO_3_MPL_L"; //PAB   443;BYTE;

      L     "DB_HR".PBanHAWE_alt.OB_SP_P_SOLL_ST_4_MPL_H;
      T     "OB_HCD_SV_CL_PO_4_MPL_H"; //PAB   444;BYTE;

      L     "DB_HR".PBanHAWE_alt.OB_SP_P_SOLL_ST_4_MPL_L;
      T     "OB_HCD_SV_CL_PO_4_MPL_L"; //PAB   445;BYTE;

      L     "DB_HR".PBanHAWE_alt.OB_SP_STATE_ST_1_RPL;
      T     "OB_HCD_STATE_CL_PO_1_SST"; //PAB   446;BYTE;

      L     "DB_HR".PBanHAWE_alt.OB_SP_STATE_ST_2_RPL;
      T     "OB_HCD_STATE_CL_PO_2_SST"; //PAB   447;BYTE;

      L     "DB_HR".PBanHAWE_alt.OB_SP_STATE_ST_3_RPL;
      T     "OB_HCD_STATE_CL_PO_3_SST"; //PAB   448;BYTE;

      L     "DB_HR".PBanHAWE_alt.OB_SP_STATE_ST_4_RPL;
      T     "OB_HCD_STATE_CL_PO_4_SST"; //PAB   449;BYTE;

      L     "DB_HR".PBanHAWE_alt.OB_SP_STATE_ST_1_MPL;
      T     "OB_HCD_STATE_CL_PO_1_MPL"; //PAB   450;BYTE;

      L     "DB_HR".PBanHAWE_alt.OB_SP_STATE_ST_2_MPL;
      T     "OB_HCD_STATE_CL_PO_2_MPL"; //PAB   451;BYTE;

      L     "DB_HR".PBanHAWE_alt.OB_SP_STATE_ST_3_MPL;
      T     "OB_HCD_STATE_CL_PO_3_MPL"; //PAB   452;BYTE;

      L     "DB_HR".PBanHAWE_alt.OB_SP_STATE_ST_4_MPL;
      T     "OB_HCD_STATE_CL_PO_4_MPL"; //PAB   453;BYTE;

      L     "DB_HR".PBanHAWE_alt.OB_SP_FUNKTION_MPL_RPL;
      T     "OB_HCD_FCT_MPL_SST"; //PAB   454;BYTE;

      L     "DB_HR".PBanHAWE_alt.OB_SP_DIAGNOSE_MPL_RPL;
      T     "OB_HCD_DIAG_MPL_SST"; //PAB   455;BYTE;

      L     "DB_HR".PBanHAWE_alt.OB_SP_P_TOL_DRUCH_ERREIC;
      T     "OB_HCD_TOL_VAL_PRE_REA"; //PAB   456;BYTE;

      L     "DB_HR".PBanHAWE_alt.OB_SP_P_TOL_NACHREGELN;
      T     "OB_HCD_TOL_VAL_READJUST"; //PAB   457;BYTE;

      L     "DB_HR".PBanHAWE_alt.OB_SP_P_TOL_NOTAUS;
      T     "OB_HCD_TOL_VAL_EMSTP"; //PAB   458;BYTE;

      L     "DB_HR".PBanHAWE_alt.OB_SP_DELTA_STEUERUNG;
      T     "OB_HCD_DELTA_CONTROL"; //PAB   459;BYTE;

      L     "DB_HR".PBanHAWE_alt.OB_SP_DELTA_REGELUNG;
      T     "OB_HCD_DELTA_REGULATION"; //PAB   460;BYTE;

      L     "DB_HR".PBanHAWE_alt.OB_SP_P_LOESEDRUCK;
      T     "OB_HCD_PRESSURE_RELEASE"; //PAB   461;BYTE;

      L     "DB_HR".PBanHAWE_alt.OB_SP_P_DRUCK_RV_OEFFNEN;
      T     "OB_HCD_PRE_RET_VALV_OPEN"; //PAB   462;BYTE;

      L     "DB_HR".PBanHAWE_alt.OB_SP_P_T_VERZ_SPANNEN;
      T     "OB_HCD_TIME_DELAY_CLAMP"; //PAB   463;BYTE;

      L     "DB_HR".PBanHAWE_alt.OB_SP_P_T_RV_OEFFNEN;
      T     "OB_HCD_RT_RET_VAL_OPEN"; //PAB   464;BYTE;

khw:  NOP   0;
NETWORK
TITLE =Ausgaenge Blum-Laser / Messeinrichtung Messtaster
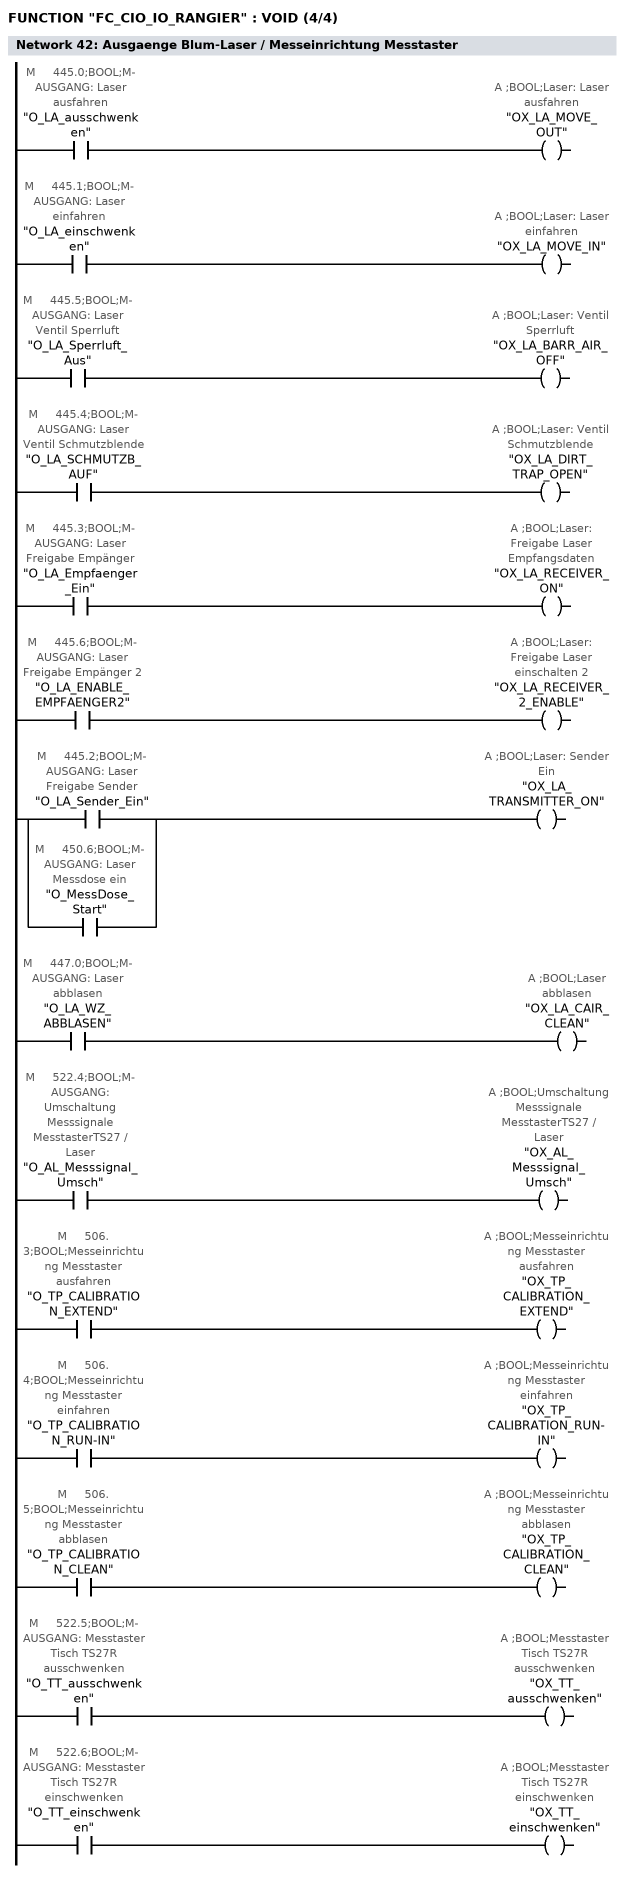

      NOP   0;

      U     "O_LA_ausschwenken"; //M     445.0;BOOL;M-AUSGANG: Laser ausfahren
      =     "OX_LA_MOVE_OUT"; //A ;BOOL;Laser: Laser ausfahren

      U     "O_LA_einschwenken"; //M     445.1;BOOL;M-AUSGANG: Laser einfahren
      =     "OX_LA_MOVE_IN"; //A ;BOOL;Laser: Laser einfahren

      U     "O_LA_Sperrluft_Aus"; //M     445.5;BOOL;M-AUSGANG: Laser Ventil Sperrluft
      =     "OX_LA_BARR_AIR_OFF"; //A ;BOOL;Laser: Ventil Sperrluft

      U     "O_LA_SCHMUTZB_AUF"; //M     445.4;BOOL;M-AUSGANG: Laser Ventil Schmutzblende
      =     "OX_LA_DIRT_TRAP_OPEN"; //A ;BOOL;Laser: Ventil Schmutzblende

      U     "O_LA_Empfaenger_Ein"; //M     445.3;BOOL;M-AUSGANG: Laser Freigabe Empänger
      =     "OX_LA_RECEIVER_ON"; //A ;BOOL;Laser: Freigabe Laser Empfangsdaten

      U     "O_LA_ENABLE_EMPFAENGER2"; //M     445.6;BOOL;M-AUSGANG: Laser Freigabe Empänger 2
      =     "OX_LA_RECEIVER_2_ENABLE"; //A ;BOOL;Laser: Freigabe Laser einschalten 2

      U     "O_LA_Sender_Ein"; //M     445.2;BOOL;M-AUSGANG: LaserFreigabe Sender
      O     "O_MessDose_Start"; //M     450.6;BOOL;M-AUSGANG: Laser Messdose ein
      =     "OX_LA_TRANSMITTER_ON"; //A ;BOOL;Laser: Sender Ein

      U     "O_LA_WZ_ABBLASEN"; //M     447.0;BOOL;M-AUSGANG: Laser abblasen
      =     "OX_LA_CAIR_CLEAN"; //A ;BOOL;Laser abblasen

      U     "O_AL_Messsignal_Umsch"; //M     522.4;BOOL;M-AUSGANG: Umschaltung Messsignale MesstasterTS27 / Laser
      =     "OX_AL_Messsignal_Umsch"; //A ;BOOL;Umschaltung Messsignale MesstasterTS27 / Laser

      U     "O_TP_CALIBRATION_EXTEND"; //M     506.3;BOOL;Messeinrichtung Messtaster ausfahren
      =     "OX_TP_CALIBRATION_EXTEND"; //A ;BOOL;Messeinrichtung Messtaster ausfahren

      U     "O_TP_CALIBRATION_RUN-IN"; //M     506.4;BOOL;Messeinrichtung Messtaster einfahren
      =     "OX_TP_CALIBRATION_RUN-IN"; //A ;BOOL;Messeinrichtung Messtaster einfahren

      U     "O_TP_CALIBRATION_CLEAN"; //M     506.5;BOOL;Messeinrichtung Messtaster abblasen
      =     "OX_TP_CALIBRATION_CLEAN"; //A ;BOOL;Messeinrichtung Messtaster abblasen

      U     "O_TT_ausschwenken"; //M     522.5;BOOL;M-AUSGANG: Messtaster Tisch TS27R ausschwenken
      =     "OX_TT_ausschwenken"; //A ;BOOL;Messtaster Tisch TS27R ausschwenken

      U     "O_TT_einschwenken"; //M     522.6;BOOL;M-AUSGANG: Messtaster Tisch TS27R einschwenken
      =     "OX_TT_einschwenken"; //A ;BOOL;Messtaster Tisch TS27R einschwenken

NETWORK
TITLE =Ausgaenge Werkzeugwechsler und Werkzeugmagazin

      NOP   0;

      U     "O_WW_1_Klappe_auf"; //M     143.6;BOOL;M-AUSGANG: Werkzeugwechsler Tuer oeffnen
      =     "OX_TC_DOOR_OPEN"; //A ;BOOL;Werkzeugwechsler Tuer oeffnen

      U     "O_WW_1_Klappe_zu"; //M     146.0;BOOL;M-AUSGANG: Werkzeugwechsler Tuer schliessen
      =     "OX_TC_DOOR_CLOSE"; //A ;BOOL;Werkzeugwechsler Tuer schliessen

      U     "O_WW_GRF_Drehen_fast"; //M     140.2;BOOL;M-AUSGANG: Werkstueckgreifer drehen schnell
      =     "OX_TC_GRP_FAST_ROTATE"; //A ;BOOL;Werkstueckgreifer drehen schnell

      U     "O_WW_GRF_Drehen_slow"; //M     140.4;BOOL;M-AUSGANG: Werkstueckgreifer drehen langsam
      =     "OX_TC_GRP_SLOW_ROTATE"; //A ;BOOL;Werkstueckgreifer drehen langsam

      U     "O_WW_1GRF_MAG"; //M     140.6;BOOL;M-AUSGANG: Werkzeuggreifer drehen Richtung Werkzeugmagazin
      =     "OX_TC_GRP_1_TOOL_MAG"; //A ;BOOL;Werkzeuggreifer drehen Richtung Werkzeugmagazin

      U     "O_WW_1GRF_SPI"; //M     143.5;BOOL;M-AUSGANG: Werkzeuggreifer drehen Richtung Spindel
      =     "OX_TC_GRP_1_SPINDLE"; //A ;BOOL;Werkzeuggreifer drehen Richtung Spindel

      U     "O_WW_Rueck_MAG"; //M     443.7;BOOL;M-AUSGANG: Werkzeug-Rueckhalt ausfahren (verriegeln)
      =     "OX_TC_RETENTION_EXTEND"; //A ;BOOL;Werkzeug-Rueckhalt ausfahren (verriegeln)
      NOT   ;
      =     "OX_TC_RETENTION_HOME_POS"; //A ;BOOL;Werkzeug-Rueckhalt zur Grundstellung

      U     "O_WW_1_ZYL_SPI"; //M      59.2;BOOL;M-AUSGANG: Werkzeugmagazin Zylinder1 Richtung Spindel / Richtung Magazin
      =     "OX_TC_CYL_1_SPINDLE"; //A ;BOOL;Werkzeugmagazin Zylinder1 Richtung Spindel

      U     "O_WW_1_ZYL_SPI"; //M      59.2;BOOL;M-AUSGANG: Werkzeugmagazin Zylinder1 Richtung Spindel / Richtung Magazin
      =     "OX_TC_CYL_1_TOOL_MAG"; //A ;BOOL;Werkzeugmagazin Zylinder1 Richtung Magazin

      U     "O_WW_1_ZYL_GST"; //M      59.3;BOOL;M-AUSGANG: Werkzeugmagazin Zylinder1 Richtung Grundstellung
      =     "OX_TC_CYL_1_HOME_POS"; //A ;BOOL;Werkzeugmagazin Zylinder1 Richtung Grundstellung

      U     "O_WW_Hub_ZYL_in_Rein"; //M     444.1;BOOL;M-AUSGANG: Werkzeugreinigung zur Stellung Reinigen
      =     "OX_TC_CLEAN_EXTEND"; //A ;BOOL;Werkzeugreinigung zur Stellung Reinigen

      UN    "O_WW_Hub_ZYL_in_Rein"; //M     444.1;BOOL;M-AUSGANG: Werkzeugreinigung zur Stellung Reinigen
      =     "OX_TC_CLEAN_HOME_POS"; //A ;BOOL;Werkzeugreinigung zur Grundstellung

      O     "O_WM_WZ_ZYL_RELEASE"; //M     459.1;BOOL;M-AUSGANG: Pneumatikzylinder Verriegelung Werkzeug loesen
      =     "OX_TM_TOOL_CYL_UNLOCK"; //A ;BOOL;Pneumatikzylinder Verriegelung Werkzeug loesen

      O     "O_WM_WZ_ZYL_RELEASE2"; //M     459.3;BOOL;M-AUSGANG: Pneumatikzylinder Verriegelung 2 Werkzeug loesen
      =     "O_WM_WZ_ZYL_RELEASE2"; //M     459.3;BOOL;M-AUSGANG: Pneumatikzylinder Verriegelung 2 Werkzeug loesen

      U     "O_WM_WZ_ZYL_CLAMP"; //M     459.0;BOOL;M-AUSGANG: Pneumatikzyl. Verriegelung WZ klemmen
      =     "OX_TM_TOOL_CYL_LOCK"; //A ;BOOL;Pneumatikzyl. Verriegelung WZ klemmen

      U     "O_WM_Freigabe_re_li"; //M     501.6;BOOL;M-AUSGANG: Freigabe Werkzeugmagazin
      =     "OX_WM_Freigabe_re_li"; //A ;BOOL;Freigabe Werkzeugmagazin

      U     "O_WM_Freigabe_re_li"; //M     501.6;BOOL;M-AUSGANG: Freigabe Werkzeugmagazin
      =     "OX_TM_RELEASE"; //A ;BOOL;Werkzeugmagazin freigeben

      U     "M_SBH_AKTIV_MAGAZIN"; //M     539.2;BOOL;SAFETY: SBH aktiv -> Freigabe Magazintüre entriegeln
      =     "OX_WM_Beladung_entr_auf"; //A ;BOOL;Freigabe Magnetverriegelung Fenster Werkzeugbestückung (Lampe)

      U     "M_SBH_AKTIV_MAGAZIN"; //M     539.2;BOOL;SAFETY: SBH aktiv -> Freigabe Magazintüre entriegeln
      =     "OX_TM_TLOAD_WDOW_UNLOCK"; //A ;BOOL;Fenster Rüstplatz entriegeln

      U     "O_WM_WZ_STAT_einlegen"; //M     197.6;BOOL;M-AUSGANG: WZV: Lampe TIN (Werkzeug einlegen)
      =     "OX_WM_WZ_STAT_einlegen"; //A ;BOOL;WZV: Lampe TIN (Werkzeug einlegen)

      U     "O_WM_WZ_STAT_einlegen"; //M     197.6;BOOL;M-AUSGANG: WZV: Lampe TIN (Werkzeug einlegen)
      =     "OX_TM_TLOAD_TIN_H"; //A ;BOOL;Meldung Werkzeug einlegen

      U     "O_WM_WZ_STAT_entnehmen"; //M     197.7;BOOL;M-AUSGANG: WZV: Lampe TOUT  (Werkzeug entnehmen)
      =     "OX_WM_WZ_STAT_entnehmen"; //A ;BOOL;WZV: Lampe TOUT  (Werkzeug entnehmen)

      U     "O_WM_WZ_STAT_entnehmen"; //M     197.7;BOOL;M-AUSGANG: WZV: Lampe TOUT  (Werkzeug entnehmen)
      =     "OX_TM_TLOAD_TOUT_H"; //A ;BOOL;Meldung Werkzeug entnehmen

      U     "O_TM_TPU_AIR_CLEANING"; //M     524.4;BOOL;M-AUSGANG: Druckluftreinigung der Transporteinheit einschalten
      O     "O_TC_TL_BRUSH_CLEAN"; //M    2031.1;BOOL;M-AUSGANG: Buerste Reinigung Werkzeugkegel
      =     "OX_TC_TL_BRUSH_CLEAN"; //A ;BOOL;Antrieb Buerste Reinigung Werkzeugkegel

      U     "O_TC_ENABLE_BRUSH_CLEAN"; //M    2030.7;BOOL;M-AUSGANG: Freigabe Positionierung Reinigung
      =     "OX_TC_ENABLE_BRUSH_CLEAN"; //A ;BOOL;Freigabe Positionierung Reinigung

      U     "O_WM_MAG_Linkslauf"; //M     436.1;BOOL;M-AUSGANG: Werkzeugmagazin Linkslauf
      =     "OX_TM_COUNTCLOCKWISE"; //A ;BOOL;Werkzeugmagazin Linkslauf

      U     "O_WM_MAG_Rechtslauf"; //M     436.0;BOOL;M-AUSGANG: Werkzeugmagazin Rechtslauf
      =     "OX_TM_CLOCKWISE"; //A ;BOOL;Werkzeugmagazin Rechtslauf

      U     "O_WW_GRF_ENTRIEGELN"; //M     299.1;BOOL;M-AUSGANG: Verriegelung Werkzeuggreifer entriegeln
      =     "OX_WW_GRF_ENTRIEGELN"; //A ;BOOL;Verriegelung Werkzeuggreifer entriegeln

      U     "O_TM_TPU_GET_TOOL"; //M     523.0;BOOL;M-AUSGANG: Transporteinheit auf Werkzeugkegel fahren
      =     "OX_TM_TPU_GET_TOOL"; //A ;BOOL;Transporteinheit auf Werkzeugkegel fahren

      U     "O_TM_TPU_RELEASE_TOOL"; //M     523.2;BOOL;M-AUSGANG: Transporteinheit vom Werkzeugkegel wegfahren
      =     "OX_TM_TPU_RELEASE_TOOL"; //A ;BOOL;Transporteinheit vom Werkzeugkegel wegfahren

      U     "O_TM_TPU_TRANSFERPOS"; //M     523.4;BOOL;M-AUSGANG: Transporteinheit zu Übergabeposition fahren
      =     "OX_TM_TPU_TRANSFERPOS"; //A ;BOOL;Transporteinheit zu Übergabeposition fahren

      U     "O_TM_TPU_MAGAZINPOS"; //M     523.6;BOOL;M-AUSGANG: Transporteinheit zur Magazinposition fahren
      =     "OX_TM_TPU_MAGAZINPOS"; //A ;BOOL;Transporteinheit zur Magazinposition fahren

      U     "O_TM_MAG_TOOL_UNLOCK"; //M     524.0;BOOL;M-AUSGANG: Werkzeug an Magazinposition entriegeln
      =     "OX_TM_MAG_TOOL_UNLOCK"; //A ;BOOL;Werkzeug an Magazinposition entriegeln

      U     "O_TM_MAG_TOOL_LOCK"; //M     524.2;BOOL;M-AUSGANG: Werkzeug an Magazinposition verriegeln
      =     "OX_TM_MAG_TOOL_LOCK"; //A ;BOOL;Werkzeug an Magazinposition verriegeln

      U     "O_TM_TPU_AIR_CLEANING"; //M     524.4;BOOL;M-AUSGANG: Druckluftreinigung der Transporteinheit einschalten
      =     "OX_TM_TPU_AIR_CLEANING"; //A ;BOOL;Druckluftreinigung der Transporteinheit einschalten

      U     "O_TM_TLOAD_TOOL_UNLOCK"; //M     524.5;BOOL;M-AUSGANG: Werkzeug am Rüstplatz entriegeln
      =     "OX_TM_TLOAD_TOOL_UNLOCK"; //A ;BOOL;Werkzeug am Rüstplatz entriegeln

      U     "O_TM_TLOAD_TOOL_LOCK"; //M     524.7;BOOL;M-AUSGANG: Werkzeug am Rüstplatz verriegeln
      =     "OX_TM_TLOAD_TOOL_LOCK"; //A ;BOOL;Werkzeug am Rüstplatz verriegeln

      U     "O_WK_MAG_AUSFAHREN"; //M     535.5;BOOL;Werkzeugtraeger ausfahren
      =     "OX_WK_ZYL_1_AUSF"; //A ;BOOL;Werkzeugträger Zylinder 1 ausfahren

      U     "O_WK_MAG_EINFAHREN"; //M     535.6;BOOL;Werkzeugtraeger einfahren
      =     "OX_WK_ZYL_1_EINFAHREN"; //A ;BOOL;Werkzeugträger Zylinder 1 einfahren

      U     "O_WK_ZYL_2_AUSF"; //M     536.1;BOOL;Werkzeugtraeger Zylinder 2 ausfahren
      =     "OX_WK_ZYL_2_AUSF"; //A ;BOOL;Werkzeugträger Zylinder 2 ausfahren

      U     "O_WK_ZYL_2_EINFAHREN"; //M     536.2;BOOL;Werkzeugtraeger Zylinder 2 einfahren
      =     "OX_WK_ZYL_2_EINFAHREN"; //A ;BOOL;Werkzeugträger Zylinder 2 einfahren

      U     "O_WK_KLAPPE_AUF"; //M     536.5;BOOL;Werkzeugklappe oeffnen
      =     "OX_WK_KLAPPE_AUF"; //A ;BOOL;Werkzeugklappe oeffnen

      U     "O_WK_KLAPPE_ZU"; //M     536.6;BOOL;Werkzeugklappe schliessen
      =     "OX_WK_KLAPPE_ZU"; //A ;BOOL;Werkzeugklappe schliessen

      U     "O_TM_PUMP"; //M    2030.5;BOOL;M-AUSGANG: Hebepumpe Werkzeugmagazin (55/65H)
      =     "OX_TM_PUMP"; //A ;BOOL;Hebepumpe Werkzeugmagazin (55/65H)

      U     "O_TC_MAGAZINPOS"; //M     634.5;BOOL;
      =     "OX_TC_MAGAZINPOS"; //A ;BOOL;

      U     "O_TC_SPIPOS"; //M     634.6;BOOL;
      =     "OX_TC_SPIPOS"; //A ;BOOL;
NETWORK
TITLE =Ausgänge Option Teepack
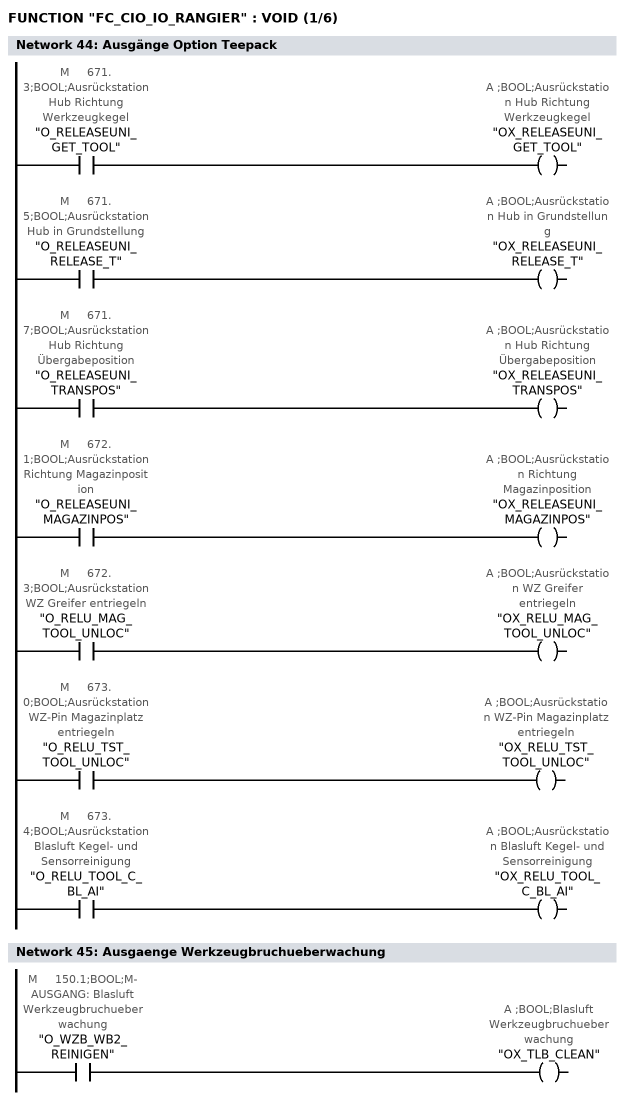

      U     "O_RELEASEUNI_GET_TOOL"; //M     671.3;BOOL;Ausrückstation Hub Richtung Werkzeugkegel
      =     "OX_RELEASEUNI_GET_TOOL"; //A ;BOOL;Ausrückstation Hub Richtung Werkzeugkegel

      U     "O_RELEASEUNI_RELEASE_T"; //M     671.5;BOOL;Ausrückstation Hub in Grundstellung
      =     "OX_RELEASEUNI_RELEASE_T"; //A ;BOOL;Ausrückstation Hub in Grundstellung

      U     "O_RELEASEUNI_TRANSPOS"; //M     671.7;BOOL;Ausrückstation Hub Richtung Übergabeposition
      =     "OX_RELEASEUNI_TRANSPOS"; //A ;BOOL;Ausrückstation Hub Richtung Übergabeposition

      U     "O_RELEASEUNI_MAGAZINPOS"; //M     672.1;BOOL;Ausrückstation Richtung Magazinposition
      =     "OX_RELEASEUNI_MAGAZINPOS"; //A ;BOOL;Ausrückstation Richtung Magazinposition

      U     "O_RELU_MAG_TOOL_UNLOC"; //M     672.3;BOOL;Ausrückstation WZ Greifer entriegeln
      =     "OX_RELU_MAG_TOOL_UNLOC"; //A ;BOOL;Ausrückstation WZ Greifer entriegeln

      U     "O_RELU_TST_TOOL_UNLOC"; //M     673.0;BOOL;Ausrückstation WZ-Pin Magazinplatz entriegeln
      =     "OX_RELU_TST_TOOL_UNLOC"; //A ;BOOL;Ausrückstation WZ-Pin Magazinplatz entriegeln

      U     "O_RELU_TOOL_C_BL_AI"; //M     673.4;BOOL;Ausrückstation Blasluft Kegel- und Sensorreinigung
      =     "OX_RELU_TOOL_C_BL_AI"; //A ;BOOL;Ausrückstation Blasluft Kegel- und Sensorreinigung
NETWORK
TITLE =Ausgaenge Werkzeugbruchueberwachung

      NOP   0;

      U     "O_WZB_WB2_REINIGEN"; //M     150.1;BOOL;M-AUSGANG: Blasluft Werkzeugbruchueberwachung
      =     "OX_TLB_CLEAN"; //A ;BOOL;Blasluft Werkzeugbruchueberwachung
NETWORK
TITLE =Ausgaenge Palettenwechsler
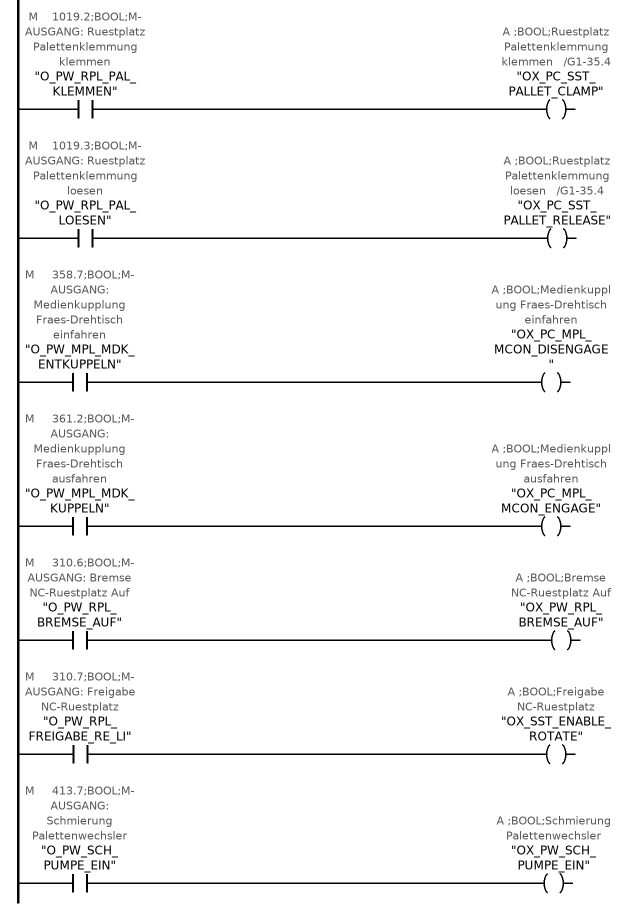

      NOP   0;

      U     "O_PC_PAL_CAR_DOWN"; //M     435.7;BOOL;M-AUSGANG: Takttisch Palettenträger senken
      =     "OX_PC_PAL_CAR_DOWN"; //A ;BOOL;Takttisch Palettenträger senken

      U     "O_4_Klem_Bremse_Auf"; //M     433.5;BOOL;M-AUSGANG: 4.Achse Klemmung lösen
      =     "OX_PC_PAL_CAR_UP"; //A ;BOOL;Takttisch Palettenträger heben

      U     "O_SP_MPL_ENTKUPPELN"; //M     356.4;BOOL;M-AUSGANG: SpannHydraulik Maschinenplatz entkuppeln
      =     "OX_HCD_MPL_DISENGAGE"; //A ;BOOL;Hydraulik Maschinenplatz Kupplung abkuppeln   /H4-05.3

      U     "O_SP_MPL_KUPPELN"; //M     356.5;BOOL;M-AUSGANG: SpannHydraulik Maschinenplatz kuppeln
      =     "OX_HCD_MPL_ENGAGE"; //A ;BOOL;Hydraulik Maschinenplatz Kupplung ankuppeln   /H4-05.3

      U     "O_SP_RPL_ENTKUPPELN"; //M     357.5;BOOL;M-AUSGANG: SpannHydraulik Rüstplatz entkuppeln
      =     "OX_HCD_SST_DISENGAGE"; //A ;BOOL;Hydraulik Rüstplatz Kupplung abkuppeln   /H4-06.3

      U     "O_SP_RPL_KUPPELN"; //M     357.6;BOOL;M-AUSGANG: SpannHydraulik Rüstplatz kuppeln
      =     "OX_HCD_SST_ENGAGE"; //A ;BOOL;Hydraulik Rüstplatz Kupplung ankuppeln   /H4-06.3

      U     "O_PW_KLE_klemmen"; //M     438.4;BOOL;M-AUSGANG: Palette auf Tisch spannen
      =     "OX_PC_MPL_PALLET_CLAMP"; //A ;BOOL;Palette auf Tisch spannen

      U     "O_PW_KLE_loesen"; //M     438.3;BOOL;M-AUSGANG: Palette auf Tisch lösen
      =     "OX_PC_MPL_PALLET_RELEASE"; //A ;BOOL;Palette auf Tisch lösen

      U     "O_PW_0_Grad_Drehen"; //M     438.7;BOOL;M-AUSGANG: Palettenwechsler schwenken 0 Grad Position
      =     "OX_PW_0_Grad_Drehen"; //A ;BOOL;Palettenwechsler schwenken 0 Grad Position

      U     "O_PW_180_Grad_Drehen"; //M     439.0;BOOL;M-AUSGANG: Palettenwechsler schwenken 180 Grad Position
      =     "OX_PW_180_Grad_Drehen"; //A ;BOOL;Palettenwechsler schwenken 180 Grad Position

      U     "O_PW_Hub_senken"; //M     438.5;BOOL;M-AUSGANG: Palettenwechsler nach unten
      =     "OX_PC_LIFT_DOWN"; //A ;BOOL;Palettenwechsler nach unten

      U     "O_PW_Hub_heben"; //M     438.6;BOOL;M-AUSGANG: Palettenwechsler nach oben
      =     "OX_PC_LIFT_UP"; //A ;BOOL;Palettenwechsler nach oben

      U     "O_PW_HUB_2_HEBEN"; //M     414.2;BOOL;M-AUSGANG: Palettenwechsler Hubeinheit nach oben schnell
      =     "OX_PC_LIFT_FAST_UP"; //A ;BOOL;Hubeinheit Palettenwechsler schnell nach oben

      U     "O_PW_HUB_2_SENKEN"; //M     414.3;BOOL;M-AUSGANG: Palettenwechsler Hubeinheit nach unten schnell
      =     "OX_PC_LIFT_FAST_DOWN"; //A ;BOOL;Hubeinheit Palettenwechsler schnell nach unten

      U     "O_PW_SPANNKONEN_ABBLAS"; //M    1021.3;BOOL;M-AUSGANG: Spannkonen abblasen
      =     "OX_PC_CLAMP_CONE_BL_O"; //A ;BOOL;Palettenträger Spannstelle ausblasen

      U     "O_PW_ACHS_Bremse_auf"; //M     141.5;BOOL;M-AUSGANG: Achse 8 (PW)  Bremse lüften
      =     "OX_PW_ACHS_Bremse_auf"; //A ;BOOL;Achse 8 (PW)  Bremse lüften

      U     "O_PW_Ventil_Abfrage"; //M      15.5;BOOL;M-AUSGANG: Ventil Luftstrom Palette
      =     "OX_PC_VALVE_REQUEST"; //A ;BOOL;Palettenwechsler Ventilabfrage Luftstrom Palette

      U     "O_PW_N_VENTIL_ABFRAGE"; //M    1020.0;BOOL;M-AUSGANG: Druckluft Palettenerkennung
      =     "OX_PC_MPL_PALLET_MONITOR"; //A ;BOOL;Druckluft Palettenerkennung

      U     "M_SBH_AKTIV_RÜSTPLATZ"; //M     539.1;BOOL;SAFETY: SBH aktiv -> Freigabe Rüstplatztüre Palettenwechsler entriegeln
      =     "OX_PC_DOOR_UNLOCK"; //A ;BOOL;Magnetverriegelung Ruestplatz Palettenwechsler entriegeln

      U     "O_RPL_TUER_OEFFNEN"; //M     347.7;BOOL;M-AUSGANG: Ventil Rüstplatztür öffnen
      =     "OX_RPL_TUER_OEFFNEN"; //M    1018.4;BOOL;M-AUSGANG: Ventil Rüstplatztür öffnen

      U     "O_RPL_TUER_SCHLIESSEN"; //M     358.1;BOOL;M-AUSGANG: Ventil Rüstplatztür schließen
      =     "OX_RPL_TUER_SCHLIESSEN"; //M    1018.5;BOOL;M-AUSGANG: Ventil Rüstplatztür schließen

      U     "O_PW_RPL_PAL_KLEMMEN"; //M    1019.2;BOOL;M-AUSGANG: Ruestplatz Palettenklemmung klemmen
      =     "OX_PC_SST_PALLET_CLAMP"; //A ;BOOL;Ruestplatz Palettenklemmung klemmen   /G1-35.4

      U     "O_PW_RPL_PAL_LOESEN"; //M    1019.3;BOOL;M-AUSGANG: Ruestplatz Palettenklemmung loesen
      =     "OX_PC_SST_PALLET_RELEASE"; //A ;BOOL;Ruestplatz Palettenklemmung loesen   /G1-35.4

      U     "O_PW_MPL_MDK_ENTKUPPELN"; //M     358.7;BOOL;M-AUSGANG: Medienkupplung Fraes-Drehtisch einfahren
      =     "OX_PC_MPL_MCON_DISENGAGE"; //A ;BOOL;Medienkupplung Fraes-Drehtisch einfahren

      U     "O_PW_MPL_MDK_KUPPELN"; //M     361.2;BOOL;M-AUSGANG: Medienkupplung Fraes-Drehtisch ausfahren
      =     "OX_PC_MPL_MCON_ENGAGE"; //A ;BOOL;Medienkupplung Fraes-Drehtisch ausfahren

      U     "O_PW_RPL_BREMSE_AUF"; //M     310.6;BOOL;M-AUSGANG: Bremse NC-Ruestplatz Auf
      =     "OX_PW_RPL_BREMSE_AUF"; //A ;BOOL;Bremse NC-Ruestplatz Auf

      U     "O_PW_RPL_FREIGABE_RE_LI"; //M     310.7;BOOL;M-AUSGANG: Freigabe NC-Ruestplatz
      =     "OX_SST_ENABLE_ROTATE"; //A ;BOOL;Freigabe NC-Ruestplatz

      U     "O_PW_SCH_PUMPE_EIN"; //M     413.7;BOOL;M-AUSGANG: Schmierung Palettenwechsler
      =     "OX_PW_SCH_PUMPE_EIN"; //A ;BOOL;Schmierung Palettenwechsler
NETWORK
TITLE =Ausgaenge Spaenefoerderer
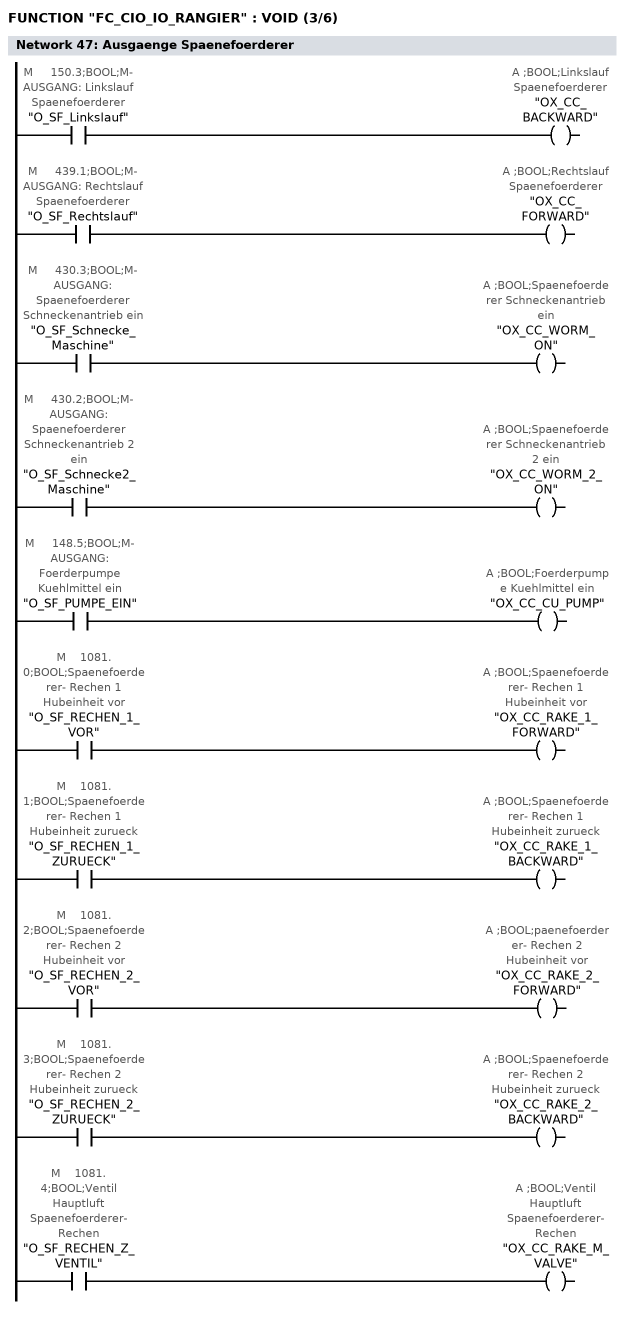

      NOP   0;

      U     "O_SF_Linkslauf"; //M     150.3;BOOL;M-AUSGANG: Linkslauf Spaenefoerderer
      =     "OX_CC_BACKWARD"; //A ;BOOL;Linkslauf Spaenefoerderer

      U     "O_SF_Rechtslauf"; //M     439.1;BOOL;M-AUSGANG: Rechtslauf Spaenefoerderer
      =     "OX_CC_FORWARD"; //A ;BOOL;Rechtslauf Spaenefoerderer

      U     "O_SF_Schnecke_Maschine"; //M     430.3;BOOL;M-AUSGANG: Spaenefoerderer Schneckenantrieb ein
      =     "OX_CC_WORM_ON"; //A ;BOOL;Spaenefoerderer Schneckenantrieb ein

      U     "O_SF_Schnecke2_Maschine"; //M     430.2;BOOL;M-AUSGANG: Spaenefoerderer Schneckenantrieb 2 ein
      =     "OX_CC_WORM_2_ON"; //A ;BOOL;Spaenefoerderer Schneckenantrieb 2 ein

      U     "O_SF_PUMPE_EIN"; //M     148.5;BOOL;M-AUSGANG: Foerderpumpe Kuehlmittel ein
      =     "OX_CC_CU_PUMP"; //A ;BOOL;Foerderpumpe Kuehlmittel ein

      U     "O_SF_RECHEN_1_VOR"; //M    1081.0;BOOL;Spaenefoerderer- Rechen 1 Hubeinheit vor
      =     "OX_CC_RAKE_1_FORWARD"; //A ;BOOL;Spaenefoerderer- Rechen 1 Hubeinheit vor

      U     "O_SF_RECHEN_1_ZURUECK"; //M    1081.1;BOOL;Spaenefoerderer- Rechen 1 Hubeinheit zurueck
      =     "OX_CC_RAKE_1_BACKWARD"; //A ;BOOL;Spaenefoerderer- Rechen 1 Hubeinheit zurueck

      U     "O_SF_RECHEN_2_VOR"; //M    1081.2;BOOL;Spaenefoerderer- Rechen 2 Hubeinheit vor
      =     "OX_CC_RAKE_2_FORWARD"; //A ;BOOL;paenefoerderer- Rechen 2 Hubeinheit vor

      U     "O_SF_RECHEN_2_ZURUECK"; //M    1081.3;BOOL;Spaenefoerderer- Rechen 2 Hubeinheit zurueck
      =     "OX_CC_RAKE_2_BACKWARD"; //A ;BOOL;Spaenefoerderer- Rechen 2 Hubeinheit zurueck

      U     "O_SF_RECHEN_Z_VENTIL"; //M    1081.4;BOOL;Ventil Hauptluft Spaenefoerderer-Rechen
      =     "OX_CC_RAKE_M_VALVE"; //A ;BOOL;Ventil Hauptluft Spaenefoerderer-Rechen

NETWORK
TITLE =Ausgaenge Fraes-Drehtisch
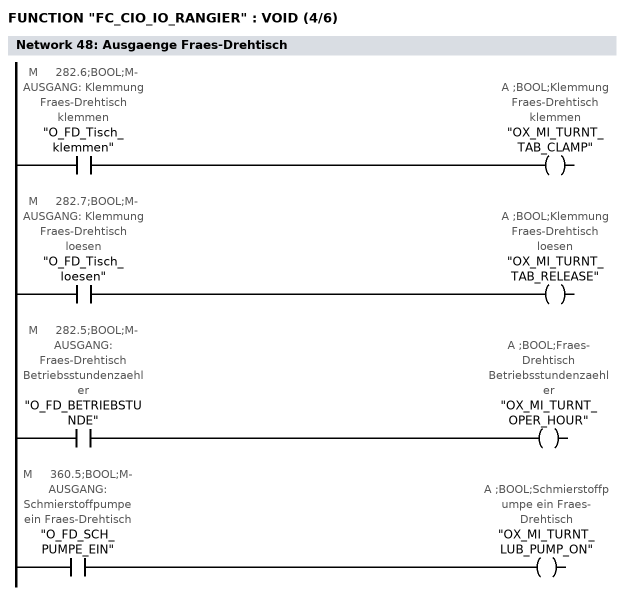

      NOP   0;

      U     "O_FD_Tisch_klemmen"; //M     282.6;BOOL;M-AUSGANG: Klemmung Fraes-Drehtisch klemmen
      =     "OX_MI_TURNT_TAB_CLAMP"; //A ;BOOL;Klemmung Fraes-Drehtisch klemmen

      U     "O_FD_Tisch_loesen"; //M     282.7;BOOL;M-AUSGANG: Klemmung Fraes-Drehtisch loesen
      =     "OX_MI_TURNT_TAB_RELEASE"; //A ;BOOL;Klemmung Fraes-Drehtisch loesen

      U     "O_FD_BETRIEBSTUNDE"; //M     282.5;BOOL;M-AUSGANG: Fraes-Drehtisch Betriebsstundenzaehler
      =     "OX_MI_TURNT_OPER_HOUR"; //A ;BOOL;Fraes-Drehtisch Betriebsstundenzaehler

      U     "O_FD_SCH_PUMPE_EIN"; //M     360.5;BOOL;M-AUSGANG: Schmierstoffpumpe ein Fraes-Drehtisch
      =     "OX_MI_TURNT_LUB_PUMP_ON"; //A ;BOOL;Schmierstoffpumpe ein Fraes-Drehtisch
NETWORK
TITLE =Ausgaenge Konzern-Kuehlmittelanlage
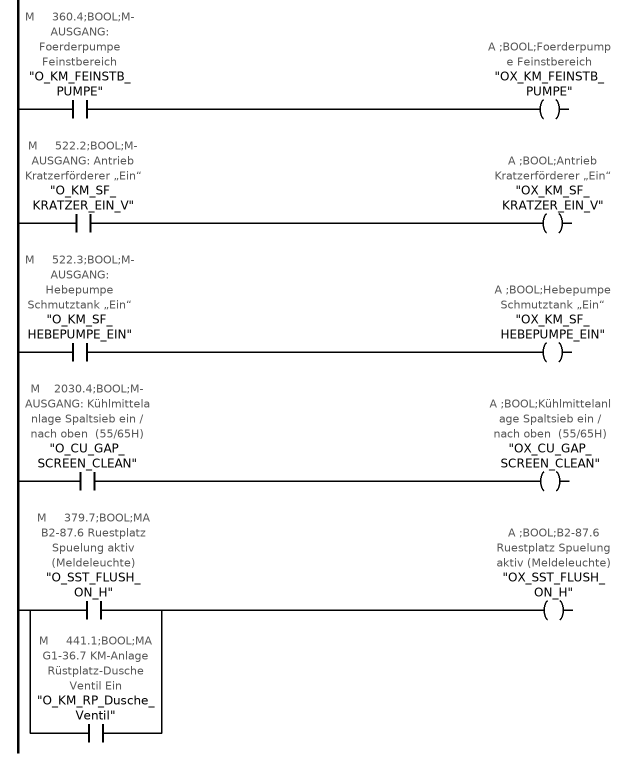

      U     "O_KM_M8_Ein"; //M     434.1;BOOL;M-AUSGANG: Pumpe Kühlmittel 1 'Ein' (M8)
      =     "OX_CU_M8"; //A ;BOOL;Pumpe Kühlmittel 1 'Ein' (M8)

      U     "O_KM_DRUCK2_M7_EIN"; //M     283.0;BOOL;M-AUSGANG: Hochdruckpumpe Kuehlmittel 2 80 bar
      =     "OX_CU_M7_STAGE_2"; //A ;BOOL;Hochdruckpumpe Kuehlmittel 2 80 bar

      U     "O_KM_Spuelpumpe_ein"; //M     443.3;BOOL;M-AUSGANG: Spaenespuelung 'Ein'
      =     "OX_CU_FLUSH_CABIN"; //A ;BOOL;Spaenespuelung 'Ein'

      U     "O_KM_TPF_MOTOR_EIN"; //M     127.2;BOOL;M-AUSGANG: Motor Ein Papierbandfilter
      =     "OX_CU_PAPER_MOVE"; //A ;BOOL;Motor Ein Papierbandfilter

      U     "O_KM_Spruehpistole_ein"; //M     439.2;BOOL;M-AUSGANG: Pumpe Kühlmittel Spülpistole
      =     "OX_CU_FLUSH_PISTOL"; //A ;BOOL;Pumpe Kühlmittel Spülpistole

      U     "DB_PLC_MD_DB20".UDHex._28_Bit6_FLUSH_JET;
      U     "O_KM_Spuelpumpe_ein"; //M     443.3;BOOL;M-AUSGANG: Spaenespuelung 'Ein'
      =     "OX_CU_FLUSH_JETS_ON"; //A ;BOOL;Ansteuerung Spuelung Spruehsystem

      U     "O_KM_Pumpe_Dach"; //M     443.2;BOOL;M-AUSGANG: Spaenespuelung Dach
      O     "O_KM_Pumpe_Dach2"; //M     443.5;BOOL;M-AUSGANG: Spaenespuelung 2 Dach
      =     "OX_CU_FLUSH_ROOF_ON"; //A ;BOOL;Ansteuerung Spuelung Dach

// Bei KSA1 gibt es nur die Klauenspülung die Dachspülungen entfallen
      U     "O_KM_Pumpe_Dach"; //M     443.2;BOOL;M-AUSGANG: Spaenespuelung Dach
      O     "O_KM_Pumpe_Dach2"; //M     443.5;BOOL;M-AUSGANG: Spaenespuelung 2 Dach
      =     "OX_CU_FLUSCH_PUMP_PC"; //A ;BOOL;Klauenspülung während PW ein

      U     "O_KM_Pumpe_Dach"; //M     443.2;BOOL;M-AUSGANG: Spaenespuelung Dach
      O     "O_KM_Pumpe_Dach2"; //M     443.5;BOOL;M-AUSGANG: Spaenespuelung 2 Dach
      O     ;
      U     "DB_PLC_MD_DB20".UDHex._28_Bit6_FLUSH_JET;
      U     "O_KM_Spuelpumpe_ein"; //M     443.3;BOOL;M-AUSGANG: Spaenespuelung 'Ein'
      =     "OX_CU_FLUSH_ROOF"; //A ;BOOL;Pumpe Spaenespuelung Dach

      U     "O_PW_Ventil_Tischspuel"; //M      15.7;BOOL;M-AUSGANG: IKZ-Pumpe ein für Tischspuelung
      =     "OX_PC_TABLE_FLUSH"; //A ;BOOL;Ventil Spänespülung Palettenwechsler

      U     "O_PW_Ventil_Tischspuel"; //M      15.7;BOOL;M-AUSGANG: IKZ-Pumpe ein für Tischspuelung
      =     "OX_CU_FLUSH_PUMP_PC"; //A ;BOOL;Pumpe Spänespülung Palettenwechsler

      U     "O_KM_M7_Ein"; //M     434.2;BOOL;M-AUSGANG: Pumpe Kühlmittel 2 'Ein' (M7)
      O     "O_KM_DRUCK1_M7_EIN"; //M     286.5;BOOL;AUSGANG: KM Druck 1 M7 ein
      UN    "O_KM_DRUCK2_M7_EIN"; //M     283.0;BOOL;M-AUSGANG: Hochdruckpumpe Kuehlmittel 2 80 bar
      O     ;
      U     "O_KM_DRUCK2_M7_EIN"; //M     283.0;BOOL;M-AUSGANG: Hochdruckpumpe Kuehlmittel 2 80 bar
      U     "DB_PLC_MD_DB20".UDHex._44_Bit5_IKZ_2DS_1PUMPE;
      =     "OX_CU_M7"; //A ;BOOL;Hochdruckpumpe Kuehlmittel 2.1

      O     "O_KM_DRUCK1_M7_EIN"; //M     286.5;BOOL;AUSGANG: KM Druck 1 M7 ein
      =     "OX_CU_M7_PRESSURE1_ON"; //A ;BOOL;

      U     "O_KM_PUMPE_FILTER_FEINB"; //M     187.7;BOOL;M-AUSGANG: Foerderpumpe Feinstbereich
      =     "OX_KM_PUMPE_FILTER_FEINB"; //A ;BOOL;Foerderpumpe Feinstbereich

      U     "O_KM_Motor_Kratzfoerd"; //M     187.2;BOOL;M-AUSGANG: Antrieb Kratzerfoerderer
      =     "OX_KM_Motor_Kratzfoerd"; //A ;BOOL;Antrieb Kratzerfoerderer

      U     "O_KM_SPRUEHPIST_RPL_EIN"; //M     286.2;BOOL;M-AUSGANG: Signalleuchte Spülpistole Rüstplatz Ein
      =     "OX_CU_FLUSH_PIST_SST_ON"; //A ;BOOL;Meldung Spuelpistole Ruestplatz ein

      U     "O_KM_FEINSTB_PUMPE"; //M     360.4;BOOL;M-AUSGANG: Foerderpumpe Feinstbereich
      =     "OX_KM_FEINSTB_PUMPE"; //A ;BOOL;Foerderpumpe Feinstbereich

      U     "O_KM_SF_KRATZER_EIN_V"; //M     522.2;BOOL;M-AUSGANG: Antrieb Kratzerförderer „Ein“
      =     "OX_KM_SF_KRATZER_EIN_V"; //A ;BOOL;Antrieb Kratzerförderer „Ein“

      U     "O_KM_SF_HEBEPUMPE_EIN"; //M     522.3;BOOL;M-AUSGANG: Hebepumpe Schmutztank „Ein“
      =     "OX_KM_SF_HEBEPUMPE_EIN"; //A ;BOOL;Hebepumpe Schmutztank „Ein“

// Kühlmittelanlage mit Spaltsieb (KSA7)
      U     "O_CU_GAP_SCREEN_CLEAN"; //M    2030.4;BOOL;M-AUSGANG: Kühlmittelanlage Spaltsieb ein / nach oben  (55/65H)
      =     "OX_CU_GAP_SCREEN_CLEAN"; //A ;BOOL;Kühlmittelanlage Spaltsieb ein / nach oben  (55/65H)

      U     "O_SST_FLUSH_ON_H"; //M     379.7;BOOL;MA B2-87.6 Ruestplatz Spuelung aktiv (Meldeleuchte)
      O     "O_KM_RP_Dusche_Ventil"; //M     441.1;BOOL;MA G1-36.7 KM-Anlage Rüstplatz-Dusche Ventil Ein
      =     "OX_SST_FLUSH_ON_H"; //A ;BOOL;B2-87.6 Ruestplatz Spuelung aktiv (Meldeleuchte)
NETWORK
TITLE =Ausgaenge Wiegenfräskopf
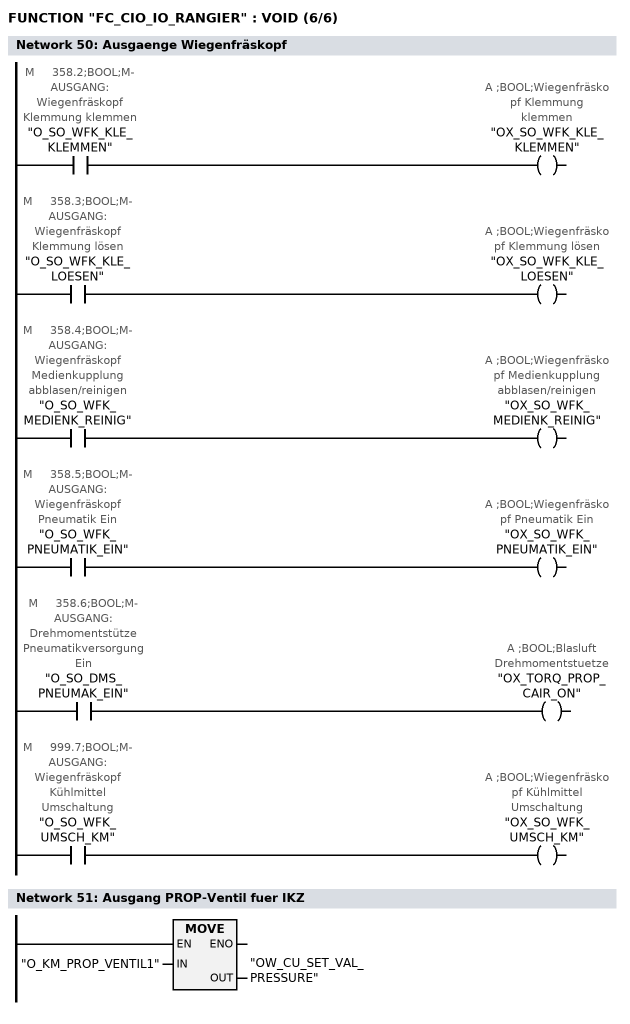

      NOP   0;

      U     "O_SO_WFK_KLE_KLEMMEN"; //M     358.2;BOOL;M-AUSGANG: Wiegenfräskopf Klemmung klemmen
      =     "OX_SO_WFK_KLE_KLEMMEN"; //A ;BOOL;Wiegenfräskopf Klemmung klemmen

      U     "O_SO_WFK_KLE_LOESEN"; //M     358.3;BOOL;M-AUSGANG: Wiegenfräskopf Klemmung lösen
      =     "OX_SO_WFK_KLE_LOESEN"; //A ;BOOL;Wiegenfräskopf Klemmung lösen

      U     "O_SO_WFK_MEDIENK_REINIG"; //M     358.4;BOOL;M-AUSGANG: Wiegenfräskopf Medienkupplung abblasen/reinigen
      =     "OX_SO_WFK_MEDIENK_REINIG"; //A ;BOOL;Wiegenfräskopf Medienkupplung abblasen/reinigen

      U     "O_SO_WFK_PNEUMATIK_EIN"; //M     358.5;BOOL;M-AUSGANG: Wiegenfräskopf Pneumatik Ein
      =     "OX_SO_WFK_PNEUMATIK_EIN"; //A ;BOOL;Wiegenfräskopf Pneumatik Ein

      U     "O_SO_DMS_PNEUMAK_EIN"; //M     358.6;BOOL;M-AUSGANG: Drehmomentstütze Pneumatikversorgung Ein
      =     "OX_TORQ_PROP_CAIR_ON"; //A ;BOOL;Blasluft Drehmomentstuetze

      U     "O_SO_WFK_UMSCH_KM"; //M     999.7;BOOL;M-AUSGANG: Wiegenfräskopf Kühlmittel Umschaltung
      =     "OX_SO_WFK_UMSCH_KM"; //A ;BOOL;Wiegenfräskopf Kühlmittel Umschaltung

NETWORK
TITLE =Ausgang PROP-Ventil fuer IKZ

      NOP   0;

      L     "O_KM_PROP_VENTIL1"; //MW    518;INT;MW-AUSGANG: Kühlmittel Hochdruck PROP-Ventil
      T     "OW_CU_SET_VAL_PRESSURE"; //AW ;WORD;Kühlmittel Hochdruck PROP-Ventil
NETWORK
TITLE =Ausgaenge Kuehlmittelanlage KNOLL

      L     "DB_PLC_MD_DB20".UDInt._019_ANWAHL_KMTL_ANLAGE;
      L     7;
      ==I   ;
      SPBN  a02;

      L     DB258.DBW    0;
      T     "OW_TUNING_CPU_KSA_0"; //PAW   300;WORD;

      L     DB258.DBW    2;
      T     "OW_TUNING_CPU_KSA_1"; //PAW   302;WORD;

      L     "DB_KMTL_KNOLL".OW_ANWAHL_DRUCKSTUFE;
      T     "OW_TUNING_CPU_KSA_2"; //PAW   304;WORD;

      L     "DB_KMTL_KNOLL".OW_KSA_KONFIGURATION;
      T     "OW_TUNING_CPU_KSA_3"; //PAW   306;WORD;

      L     "DB_KMTL_KNOLL".OW_FUNCTION_1;
      T     "OW_TUNING_CPU_KSA_4"; //PAW   308;WORD;

a02:  NOP   0;

      L     "DB_PLC_MD_DB20".UDInt._019_ANWAHL_KMTL_ANLAGE;
      L     8;
      ==I   ;
      O     "DB_PLC_MD_DB20".UDHex._25_Bit3_SOKO_Kuehlm;
      SPBN  a12;

      L     DB258.DBW    0;
      TAW   ;
      T     "OW_TUNING_CPU_KSA_0"; //PAW   300;WORD;

      L     DB258.DBW    2;
      TAW   ;
      T     "OW_TUNING_CPU_KSA_1"; //PAW   302;WORD;

      L     "DB_KMTL_KNOLL".OW_ANWAHL_DRUCKSTUFE;
      TAW   ;
      T     "OW_TUNING_CPU_KSA_2"; //PAW   304;WORD;

      L     "DB_KMTL_KNOLL".OW_KSA_KONFIGURATION;
      T     "OW_TUNING_CPU_KSA_3"; //PAW   306;WORD;

      L     "DB_KMTL_KNOLL".OW_FUNCTION_1;
      T     "OW_TUNING_CPU_KSA_4"; //PAW   308;WORD;

      L     "DB_KMTL_KNOLL".OW_PARAMETER_2;
      T     "OW_TUNING_CPU_KSA_5"; //PAW   310;WORD;

a12:  NOP   0;
NETWORK
TITLE =Ausgaenge OMRON-Regalmagazin

      U     "M_WZM_Regal_angewaehlt"; //M     354.0;BOOL;WZW: OMRON-Regalmagazin angewaehlt
      SPBN  M016;

      L     DB251.DBW    0;
      TAW   ;
      T     PAW  258;

      L     "DB_SCHNITTST_OMRON".OW_WMR_CNC_MAINCOMMAND;
      T     PAW  262;

      L     "DB_SCHNITTST_OMRON".OW_WMR_CNC_SUBCOMMAND;
      T     PAW  264;

      L     "DB_SCHNITTST_OMRON".OW_WMR_CNC_1_DATA;
      T     PAW  266;

      L     "DB_SCHNITTST_OMRON".OW_WMR_CNC_2_DATA;
      T     PAW  268;

      L     "DB_SCHNITTST_OMRON".OW_WMR_CNC_SENDEN;
      T     PAW  270;

      L     "DB_SCHNITTST_OMRON".OW_WMR_CNC_EMPFANGEN;
      T     PAW  272;

M016: NOP   0;

NETWORK
TITLE =Ausgaenge Palettenrundspeicher
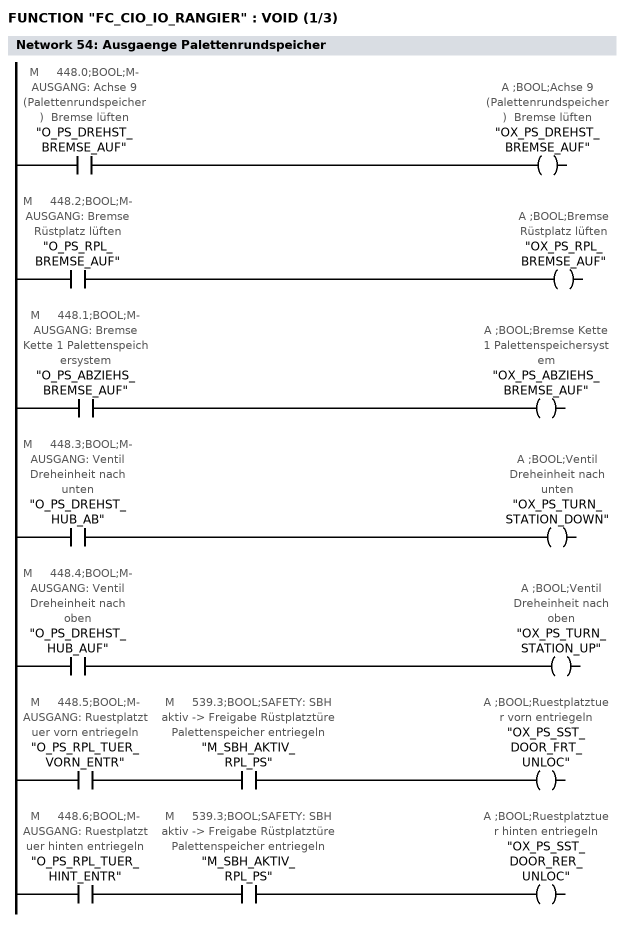

      U     "O_PS_DREHST_BREMSE_AUF"; //M     448.0;BOOL;M-AUSGANG: Achse 9 (Palettenrundspeicher)  Bremse lüften
      =     "OX_PS_DREHST_BREMSE_AUF"; //A ;BOOL;Achse 9 (Palettenrundspeicher)  Bremse lüften

      U     "O_PS_RPL_BREMSE_AUF"; //M     448.2;BOOL;M-AUSGANG: Bremse Rüstplatz lüften
      =     "OX_PS_RPL_BREMSE_AUF"; //A ;BOOL;Bremse Rüstplatz lüften

      U     "O_PS_ABZIEHS_BREMSE_AUF"; //M     448.1;BOOL;M-AUSGANG: Bremse Kette 1 Palettenspeichersystem
      =     "OX_PS_ABZIEHS_BREMSE_AUF"; //A ;BOOL;Bremse Kette 1 Palettenspeichersystem

      U     "O_PS_DREHST_HUB_AB"; //M     448.3;BOOL;M-AUSGANG: Ventil Dreheinheit nach unten
      =     "OX_PS_TURN_STATION_DOWN"; //A ;BOOL;Ventil Dreheinheit nach unten

      U     "O_PS_DREHST_HUB_AUF"; //M     448.4;BOOL;M-AUSGANG: Ventil Dreheinheit nach oben
      =     "OX_PS_TURN_STATION_UP"; //A ;BOOL;Ventil Dreheinheit nach oben

      U     "O_PS_RPL_TUER_VORN_ENTR"; //M     448.5;BOOL;M-AUSGANG: Ruestplatztuer vorn entriegeln
      U     "M_SBH_AKTIV_RPL_PS"; //M     539.3;BOOL;SAFETY: SBH aktiv -> Freigabe Rüstplatztüre Palettenspeicher entriegeln
      =     "OX_PS_SST_DOOR_FRT_UNLOC"; //A ;BOOL;Ruestplatztuer vorn entriegeln

      U     "O_PS_RPL_TUER_HINT_ENTR"; //M     448.6;BOOL;M-AUSGANG: Ruestplatztuer hinten entriegeln
      U     "M_SBH_AKTIV_RPL_PS"; //M     539.3;BOOL;SAFETY: SBH aktiv -> Freigabe Rüstplatztüre Palettenspeicher entriegeln
      =     "OX_PS_SST_DOOR_RER_UNLOC"; //A ;BOOL;Ruestplatztuer hinten entriegeln
NETWORK
TITLE =Ausgaenge EROWA / PROMOT
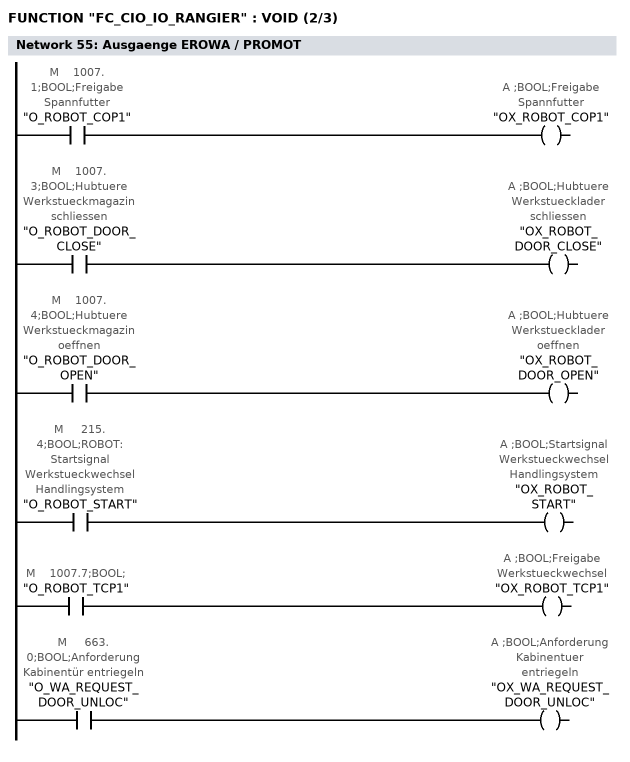

      U     "O_ROBOT_COP1"; //M    1007.1;BOOL;Freigabe Spannfutter
      =     "OX_ROBOT_COP1"; //A ;BOOL;Freigabe Spannfutter

      U     "O_ROBOT_DOOR_CLOSE"; //M    1007.3;BOOL;Hubtuere Werkstueckmagazin schliessen
      =     "OX_ROBOT_DOOR_CLOSE"; //A ;BOOL;Hubtuere Werkstuecklader schliessen

      U     "O_ROBOT_DOOR_OPEN"; //M    1007.4;BOOL;Hubtuere Werkstueckmagazin oeffnen
      =     "OX_ROBOT_DOOR_OPEN"; //A ;BOOL;Hubtuere Werkstuecklader oeffnen

      U     "O_ROBOT_START"; //M     215.4;BOOL;ROBOT: Startsignal Werkstueckwechsel Handlingsystem
      =     "OX_ROBOT_START"; //A ;BOOL;Startsignal Werkstueckwechsel Handlingsystem

      U     "O_ROBOT_TCP1"; //M    1007.7;BOOL;
      =     "OX_ROBOT_TCP1"; //A ;BOOL;Freigabe Werkstueckwechsel

      U     "O_WA_REQUEST_DOOR_UNLOC"; //M     663.0;BOOL;Anforderung Kabinentür entriegeln
      =     "OX_WA_REQUEST_DOOR_UNLOC"; //A ;BOOL;Anforderung Kabinentuer entriegeln

NETWORK
TITLE =Ausgaenge U-Achse
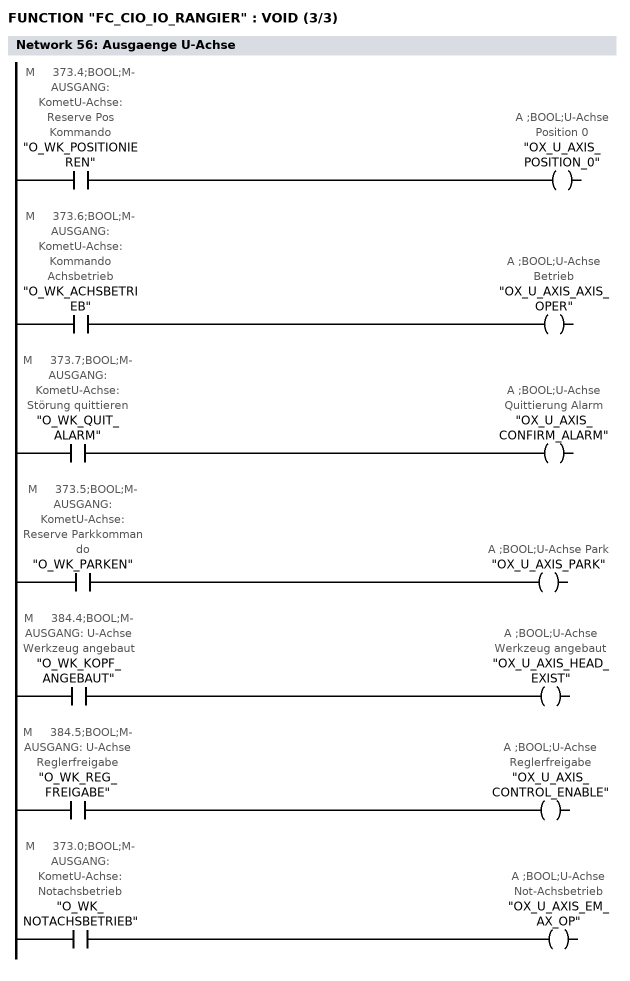

      NOP   0;

      U     "O_WK_POSITIONIEREN"; //M     373.4;BOOL;M-AUSGANG: KometU-Achse:Reserve PosKommando
      =     "OX_U_AXIS_POSITION_0"; //A ;BOOL;U-Achse Position 0

      U     "O_WK_ACHSBETRIEB"; //M     373.6;BOOL;M-AUSGANG: KometU-Achse:Kommando Achsbetrieb
      =     "OX_U_AXIS_AXIS_OPER"; //A ;BOOL;U-Achse Betrieb

      U     "O_WK_QUIT_ALARM"; //M     373.7;BOOL;M-AUSGANG: KometU-Achse:Störung quittieren
      =     "OX_U_AXIS_CONFIRM_ALARM"; //A ;BOOL;U-Achse Quittierung Alarm

      U     "O_WK_PARKEN"; //M     373.5;BOOL;M-AUSGANG: KometU-Achse:Reserve Parkkommando
      =     "OX_U_AXIS_PARK"; //A ;BOOL;U-Achse Park

      U     "O_WK_KOPF_ANGEBAUT"; //M     384.4;BOOL;M-AUSGANG: U-Achse Werkzeug angebaut
      =     "OX_U_AXIS_HEAD_EXIST"; //A ;BOOL;U-Achse Werkzeug angebaut

      U     "O_WK_REG_FREIGABE"; //M     384.5;BOOL;M-AUSGANG: U-Achse Reglerfreigabe
      =     "OX_U_AXIS_CONTROL_ENABLE"; //A ;BOOL;U-Achse Reglerfreigabe

      U     "O_WK_NOTACHSBETRIEB"; //M     373.0;BOOL;M-AUSGANG: KometU-Achse:Notachsbetrieb
      =     "OX_U_AXIS_EM_AX_OP"; //A ;BOOL;U-Achse Not-Achsbetrieb
NETWORK
TITLE =Ausgaenge Handlingsystem
//DB243 Instanz-DB "DI_FB_IF_FASTEMS"
//
//      CALL  "FB_IF_FASTEMS" , "DI_FB_IF_FASTEMS"
//       I_Reserved              :="m_null"
//       I_plc_Pallet_on_APC     :="I_PW_UPL_PAL_VORH"
//       I_plc_APC_home_position :=#t_Crane_Movement_allowed
//       I_plc_APC_A_side_out    :="DB_PW_DATA".bPW_0Grad
//       I_plc_APC_B_Side_out    :="DB_PW_DATA".bPW_180Grad
//       I_plc_Palletchangeactive:="M_PW_Aktiv"
//       I_plc_oper_or_apc_door_c:=#t_oper_or_apc_door
//       I_plc_On_line           :="M_Automatik_Betrieb"
//       I_plc_Cycle_on          :="DB_SIEM_KANAL_1".E_ProgRunn
//       I_plc_Feed_on           :=#t_Feed_on
//       I_plc_Alarm             :=#t_PLC_Fehler
//       I_FixtureonAPC          :="MX_FIXTURE_ON_APC"
//       I_FixtureReleased       :="MX_FIXTURE_RELEASED"
//       I_FixtureLocked         :="MX_Fixture_Locked"
//       I_reserveByte2Bit6      :=
//       I_reserveByte2Bit7      :=
//       I_MMS_Reserved_for_diagc:=
//       I_MMS_APC_movement_ok   :="I_FMS_APC_MOVEMENT_OK"
//       I_MMS_cycle_start       :="I_FMS_NC_START"
//       I_MMS_AutoPowerOffToMC  :="I_FMS_AUTO_POWER_OFF"
//       I_MMS_Release_Fixture   :="I_FMS_FIXTURE_RELEASE"
//       I_MMS_Reserve_1bit5     :=
//       I_MMS_Reserve_1bit6     :=
//       I_MMS_Reserve_1bit7     :=
//       I_RPC_palett_data       :=
//       I_RPC_command           :=
//
      U(    ;
      L     "DB_PLC_MD_DB20".UDInt._027_ANWAHL_HANDLINGSYST;
      L     3;
      ==I   ;
      )     ;
      O(    ;
      L     "DB_PLC_MD_DB20".UDInt._027_ANWAHL_HANDLINGSYST;
      L     8;
      ==I   ;
      )     ;
      O(    ;
      L     "DB_PLC_MD_DB20".UDInt._027_ANWAHL_HANDLINGSYST;
      L     9;
      ==I   ;
      )     ;
      SPBN  M020;


      L     DB243.DBB    0;
      T     PAB 1150; //"PAW_FMS_AW1"

      U(    ;
      L     "DB_PLC_MD_DB20".UDInt._027_ANWAHL_HANDLINGSYST;
      L     8;
      ==I   ;
      )     ;
      O(    ;
      L     "DB_PLC_MD_DB20".UDInt._027_ANWAHL_HANDLINGSYST;
      L     9;
      ==I   ;
      )     ;
      SPBN  M020;

      L     DB243.DBW    1;
      T     PAW 1151;

      L     DB243.DBW    3;
      T     PAW 1153;


M020: NOP   0;



//------------ nur für IBN-Tool, damit keine FM generiert werden ------------------
      U     "OX_FMS_PALLET_ON_APC"; //A ;BOOL;MC OUTPUT Byte 1 Bit 1
      U     "OX_FMS_CRANE_MOVE_OK"; //A ;BOOL;MC OUTPUT Byte 1 Bit 2
      U     "OX_FMS_APC_A_SIDE_OUT"; //A ;BOOL;MC OUTPUT Byte 1 Bit 3
      U     "OX_FMS_APC_B_SIDE_OUT"; //A ;BOOL;MC OUTPUT Byte 1 Bit 4
      U     "OX_FMS_PALLET_CHANGE_AKT"; //A ;BOOL;MC OUTPUT Byte 1 Bit 5
      U     "OX_FMS_APC_DOOR_CLOSED"; //A ;BOOL;MC OUTPUT Byte 1 Bit 6
      U     "OX_FMS_OM_ENABLE"; //A ;BOOL;MC OUTPUT Byte 1 Bit 7
      U     "OX_FMS_MACHINE_PGM_RUN"; //A ;BOOL;MC OUTPUT Byte 2 Bit 0
      U     "OX_FMS_CUTTING"; //A ;BOOL;MC OUTPUT Byte 2 Bit 1
      U     "OX_FMS_MACHINE_ERROR"; //A ;BOOL;MC OUTPUT Byte 2 Bit 2
      U     "OX_FMS_FIXTURE_EXIST"; //A ;BOOL;MC OUTPUT Byte 2 Bit 3
      U     "OX_FMS_FIXTURE_RELEASED"; //A ;BOOL;MC OUTPUT Byte 2 Bit 4
      =     #TEMP;
//---------------------------------------------------------------------------------

      U     "O_FMS_OM1_DISABLED"; //M    1041.1;BOOL;Betriebsart Automatik gesperrt Palettenspeichersystem
      =     "OX_FMS_OM1_DISABLED"; //A ;BOOL;Betriebsart Automatik gesperrt Palettenspeichersystem

NETWORK
TITLE =Ausgaenge Roboter-Schnittstelle - Start-Adr für DPDP-Koppler
//Übertragen auf ProfiBus-Ausgänge vom Baustein für Roboter-Schnittstelle DB701
//erfolgt im FC_ROB_MIT_RPL_MAIN mit FC_UT_IO_PROFIBUS.
//Hier wird nur die Start-Adresse definiert.
//nur für IBN-Tool, damit keine Fehlermeldung generiert wird
      SPA   R_2;
      L     "DB_CONFIG".ProfiBus.StartAdrPLC.OUT_Robot;
      T     "OW_ROBOT_0"; //PAW  1160;WORD;xx-xx.x MA Start-Adr: Roboter-Schnittstelle - DPDP-Koppler

R_2:  L     1160;
      T     "DB_CONFIG".ProfiBus.StartAdrPLC.OUT_Robot;
NETWORK
TITLE =Ausgaenge SOKO-Slave(8) DB_IN-Signale
//Nur für IBN-Tool (absoluter Sprung)
//
//Daten LESEN + SCHREIBEN erfolgt im FC_SONDER_MAIN
//wegen Kompatibilität zu alten Maschinen ist Funktion nicht in FC_CIO_IO_RANGIER
//verlegbar.
//
//SOKO-Eingänge (Daten PLC==>SOKO):
//Daten von DB171 auf Peripherie-Ausgänge PAW210...PAW241 schreiben.
//
//Bei allen SOKO-Informationen, die als BYTE oder BIT interpretiert werden,
//müssen HIGH-Byte und LOW-Byte mit TAW getauscht werden.
//
//SOKO-Slave(8)-Liste:
//swic\Pfronten\Steuerungsunabhängige Dokumente\Spezifikationen\SOKO
      SPA   SO_2;

      L     DB171.DBW    0;
      TAW   ;
      T     "OW_Tuning_CPU_0"; //PAW   210;WORD;xx-xx.x MA Datenschnittstelle Profibus(8)

      L     DB171.DBW    2;
      TAW   ;
      T     "OW_Tuning_CPU_1"; //PAW   212;WORD;xx-xx.x MA Datenschnittstelle Profibus(8)

      L     DB171.DBW    4;
      TAW   ;
      T     "OW_Tuning_CPU_2"; //PAW   214;WORD;xx-xx.x MA Datenschnittstelle Profibus(8)

      L     DB171.DBW    6;
      TAW   ;
      T     "OW_Tuning_CPU_3"; //PAW   216;WORD;xx-xx.x MA Datenschnittstelle Profibus(8)

      L     DB171.DBW    8;
      TAW   ;
      T     "OW_Tuning_CPU_4"; //PAW   218;WORD;xx-xx.x MA Datenschnittstelle Profibus(8)

      L     "DB_IN".EMW_PARAMETER_1;
      T     "OW_Tuning_CPU_C0"; //PAW   220;WORD;xx-xx.x MA Datenschnittstelle Profibus(8)

      L     "DB_IN".EMW_PARAMETER_2;
      T     "OW_Tuning_CPU_C1"; //PAW   222;WORD;xx-xx.x MA Datenschnittstelle Profibus(8)

      L     "DB_IN".EMW_PARAMETER_3;
      T     "OW_Tuning_CPU_C2"; //PAW   224;WORD;xx-xx.x MA Datenschnittstelle Profibus(8)

      L     "DB_IN".EMW_PARAMETER_4;
      T     "OW_Tuning_CPU_C3"; //PAW   226;WORD;xx-xx.x MA Datenschnittstelle Profibus(8)

      L     DB171.DBW   18;
      TAW   ;
      T     "OW_Tuning_CPU_5"; //PAW   228;WORD;xx-xx.x MA Datenschnittstelle Profibus(8)

      L     "DB_IN".EMW_FUNCTION1;
      T     "OW_Tuning_CPU_6"; //PAW   230;WORD;xx-xx.x MA Datenschnittstelle Profibus(8)

      L     DB171.DBW   22;
      TAW   ;
      T     "OW_TUNING_CPU_7"; //PAW   232;WORD;xx-xx.x MA Datenschnittstelle Profibus(8)

      L     DB171.DBW   24;
      TAW   ;
      T     "OW_TUNING_CPU_8"; //PAW   234;WORD;

SO_2: NOP   0;
NETWORK
TITLE =Ein-/Aus-Gaenge für ARTIS + Toolinspect (nur für IBN-Tool)
//nur, damit IBN-Tool keine Fehlermeldung bringt.
//Adresszuornung erfolgt in HW-Konfiguration
      SPA   ARTI;
      L     "IB_TOOL_CUT_FORCE_1_MON"; //PEB  1300;BYTE;ARTIS/Toolinspect Eingangs-Byte 1
      T     #TEMP5;

      L     0;
      T     "OB_TOOL_CUT_FORCE_1_MON"; //PAB  1300;BYTE;ARTIS/Toolinspect Ausgangs-Byte 1
      T     "OB_TOOL_CUT_FORCE_2_MON"; //PAB  1301;BYTE;ARTIS/Toolinspect Ausgangs-Byte 2
ARTI: NOP   0;
NETWORK
TITLE =Ausgaenge Nicht verwendete Ausgänge
//Ausgänge, die in der HW konfiguriert werden müssen, aber noch nicht verwendet
//werden.
      CLR   ;
      =     "BT_ET200S_4_14"; //A ;BOOL;Reserve Modul
NETWORK
TITLE =----- Ende normale Abarbeitung -----

      BEA   ;

NETWORK
TITLE =BISC_Balluf
//Wird noch  im FC 83 direkt auf PAW160 geschrieben
//Dies sind nur Dummy Merker um im IBN Tool die Fehlermeldung zu unterdrücken.
//
      L     "O_BIS_C_35"; //MW    484;WORD;Balluff
      T     "OW_BIS_C_35"; //PAW  1060;WORD;Balluff
NETWORK
TITLE =Schnelle Eingaenge

M004: L     "DB_PLC_MD_DB20".UDInt._010_ANWAHL_WERZEUGBRUCH;
      L     0;
      >I    ;
      SPBN  M018;

// Schnellabschaltung Werkzeugbruch
// Es muss von der Hardwarekonstruktion immer das EB41 verwendet werden
      L     PEB   41;
      T     "MB_Werkzeugbruch"; //MB    500;BYTE;

      U     "IX_TLB_BIT_0"; //M     500.0;BOOL;M-EINGANG: WZB Binärcodiert
      =     "I_WZB_Bit_0"; //M     339.2;BOOL;M-EINGANG: Werkzeugbruchüberwachung BCD-Zahl 1

      U     "IX_TLB_BIT_1"; //M     500.1;BOOL;M-EINGANG: WZB Binärcodiert
      =     "I_WZB_Bit_1"; //M     339.3;BOOL;M-EINGANG: Werkzeugbruchüberwachung BCD-Zahl 2

      U     "IX_TLB_BIT_2"; //M     500.2;BOOL;M-EINGANG: WZB Binärcodiert
      =     "I_WZB_Bit_2"; //M     339.4;BOOL;M-EINGANG: Werkzeugbruchüberwachung BCD-Zahl 4

      U     "IX_TLB_BIT_3"; //M     500.3;BOOL;M-EINGANG: WZB Binärcodiert
      =     "I_WZB_Bit_3"; //M     339.5;BOOL;M-EINGANG: Werkzeugbruchüberwachung BCD-Zahl 8

      U     "IX_TLB_MEASURING_END"; //M     500.4;BOOL;M-EINGANG: WZB Messung Ende
      =     "I_WZB_Messung_Ende"; //M     339.1;BOOL;M-EINGANG: Werkzeugbruchüberwachung Messwertübernahme

      U     "IX_TLB_HOME_POS"; //M     500.5;BOOL;M-EINGANG: WZB Parkstellung
      =     "I_WZB_Parkstellung"; //M     268.1;BOOL;M-EINGANG: Bruchüberwachung in Parkstellung



// Schnellabschaltung Palettenwechsler mitte
// Es muss von der Hardwarekobstruktion immer der E66.2 für "IX_PC_LIFT_MID" verwendet werden
// Ist "IX_PC_LIFT_MID" nicht in der Zuli vorhanden ist Temp8 immer null und der "I_PW_Hub_in_Mitte" wird nicht geschrieben
M018: U     "m_null";
      =     #TEMP8;

      U     "IX_PC_LIFT_MID";
      ON    "IX_PC_LIFT_MID";
      =     #TEMP8;


      U     #TEMP8;
      SPBN  kpcm;

      L     PEB   66;
      T     "MB_PERIPHERIE_E_BYTE66"; //MB   2066;BYTE;Zwischenspeicher Peripherie-Eingangsbyte 66

      O     "M_PC_LIFT_MID_PERIPH_E"; //M    2066.2;BOOL;Schneller Eingang Palettenwechsler mitte E66.2 Peripherie-Eingang
      =     "I_PW_Hub_in_Mitte"; //M      16.3;BOOL;M-EINGANG: Palettenwechsler Hub Pos. Mitte
kpcm: NOP   0;

//Bei H-Maschinen werdem die Spanner-Eingänge durch den OB35 Aufruf gelesen (Span_zu_Span_Zeit Optimierung)
      UN    "DB_CONFIG".ANWAHL_DURCH_USER_DATA.MASCHTYP_3071_AKTIV;
      SPB   Hma3;

//für eine weitere Optimierung der "Span zu Span Zeit" bei H-Maschinen mit Solutionline (55H/65H/75H und künftige)
//werden die Eingänge und Ausgänge des Werkzeugspanners in Zukunft über die entsprechenden Peripherie Ein/Ausgangsbytes
//im OB35 alle 10ms gelesen bzw. geschreiben.
//Dies setzt voraus das die E/A Belegung wie unten auch zukünftig bestand hat.
//IX_SPI_TL_CLP_RELEASED    E      63.4   Werkzeugspanner geloest / C2-03.2
//IX_SPI_TL_CLP_CLAMPED    E      63.5  Werkzeugspanner gespannt / C2-03.5
//IX_TOOL_CLAMP_CLPD_WO_TL      E63.7      Werkzeugspanner gespannt ohne Werkzeug


      L     PEB   63;
      T     "MB_PERIPHERIE_E_BYTE63";

      U     "M_WZ_SPA_GEL_PERIPH_E"; // "IX_SPI_TL_CLP_RELEASED"
      =     "I_WZ_SPA_geloest";

      U     "M_WZ_SPA_GES_PERIPH_E"; //"IX_SPI_TL_CLP_CLAMPED"
      =     "I_WZ-Spanner_Gesp_O_WZ";

      U     "M_WZ_SPA_GES_PERIPH_E"; // "IX_SPI_TL_CLP_CLAMPED"
      =     "I_WZ_SPA_gespannt";

//Abfrage ob Schalter"IX_TOOL_CLAMP_CLPD_WO_TL" vorhanden ist
      U     "m_null";
      =     #TEMP9;

      U     "IX_TOOL_CLAMP_CLPD_WO_TL";
      ON    "IX_TOOL_CLAMP_CLPD_WO_TL";
      =     #TEMP9;

      U     #TEMP9;
      SPBN  Hma3;


      U     "M_WZ_SPA_GES_OW_PERIPH_E"; //E ;BOOL;
      =     "I_WZ-Spanner_Gesp_O_WZ"; //M     338.3;BOOL;M-EINGANG: Werkzeugspanner gespannt ohne Werkzeug

      UN    "M_WZ_SPA_GES_OW_PERIPH_E"; //E ;BOOL;
      U     "M_WZ_SPA_GES_PERIPH_E"; //E ;BOOL;Werkzeugspanner gespannt
      =     "I_WZ-Spanner_Gesp_mit_WZ"; //M     307.0;BOOL;

Hma3: NOP   0;
NETWORK
TITLE =Baustein-Ende

      BEA   ;

NETWORK
TITLE =Schnelle Ausgaenge

M005: L     "DB_PLC_MD_DB20".UDInt._010_ANWAHL_WERZEUGBRUCH;
      L     0;
      >I    ;
      SPBN  M019;

// Schnellabschaltung Werkzeugbruch
// Es muss von der Hardwarekonstruktion immer der A43.6 für "OX_TLB_ENABLE" verwendet werden
      U     "O_WZB_Messung_Start"; //M     438.0;BOOL;M-AUSGANG: Werkzeugbruchüberwachung Freigabe
      =     "OX_TLB_ENABLE"; //A ;BOOL;WZB Messung Start


      L     AB    43;
      T     PAB   43;


// Schnellabschaltung Palettenwechsler mitte
// Es muss von der Hardwarekonstruktion immer der A76.0 u A76.1 für "OX_PC_LIFT_DOWN" und "OX_PC_LIFT_UP" verwendet werden
M019: U     "O_PW_Hub_senken"; //M     438.5;BOOL;M-AUSGANG: Palettenwechsler nach unten
      =     "OX_PC_LIFT_DOWN"; //A ;BOOL;Palettenwechsler nach unten

      U     "O_PW_Hub_heben"; //M     438.6;BOOL;M-AUSGANG: Palettenwechsler nach oben
      =     "OX_PC_LIFT_UP"; //A ;BOOL;Palettenwechsler nach oben

      L     AB    76;
      T     PAB   76;

//Bei H-Maschinen werdem die Spanner-Ausänge durch den OB35 Aufruf geschrieben (Span_zu_Span_Zeit Optimierung)
      UN    "DB_CONFIG".ANWAHL_DURCH_USER_DATA.MASCHTYP_3071_AKTIV;
      SPB   Hma4;

//für eine weitere Optimierung der "Span zu Span Zeit" bei H-Maschinen mit Solutionline (55H/65H/75H und künftige)
//werden die Eingänge und Ausgänge des Werkzeugspanners in Zukunft über die entsprechenden Peripherie Ein/Ausgangsbytes
//im OB35 alle 10ms gelesen bzw. geschreiben.
//Dies setzt voraus das die E/A Belegung wie unten auch zukünftig bestand hat.
//OX_SPI_TL_CLAMP_RELEASE    A      42.2  Werkzeugspanner loesen / C2-01.1
//OX_SPI_TL_CLP_CLAMP    A      32.0   Werkzeugspanner Spannen / C2-04.4

      U     "O_AL_WZ_Spanner_Loesen";
      O     "M_O_Anwahl_WZS_Man";
      =     "OX_SPI_TL_CLAMP_RELEASE";

      L     AB    42;
      T     PAB   42;

      UN    "O_AL_WZ_Spanner_Loesen";
      UN    "M_Tast_Man_WZSp";
      =     "OX_SPI_TL_CLP_CLAMP";

      L     AB    32;
      T     PAB   32;

Hma4: NOP   0;

NETWORK
TITLE =Baustein-Ende

M006: BEA   ;

END_FUNCTION

